METHOD PROTECTED OnExecute
VAR
END_VAR
out.Value := in1.Value AND in2.Value;
END_METHOD

END_FUNCTION_BLOCK

// Logic/Nodes/AND/AND_DINT
{attribute 'linkalways'} 
{attribute 'no_explicit_call' := 'This FB is a CLASS and must be accessed using methods or properties'}
{attribute 'enable_dynamic_creation'}
FUNCTION_BLOCK FINAL AND_DINT EXTENDS Node
VAR
	in1 : _DINT(0);
	in2 : _DINT(0);
	out : _DINT(0);
END_VAR

METHOD FB_init : BOOL
VAR_INPUT
	bInitRetains : BOOL; // if TRUE, the retain variables are initialized (warm start / cold start)
	bInCopyCode : BOOL;  // if TRUE, the instance afterwards gets moved into the copy code (online change)
END_VAR
AddInput('in1',THIS^.in1);
AddInput('in2',THIS^.in2);
AddOutput('out', THIS^.out);
END_METHOD

METHOD PUBLIC Clone : I_Node
VAR
	pNode : POINTER TO AND_DINT;
END_VAR
pNode := __NEW(AND_DINT);
Clone := pNode^;
END_METHOD

METHOD PROTECTED OnExecute
VAR
END_VAR
out.Value := in1.Value AND in2.Value;
END_METHOD

END_FUNCTION_BLOCK

// Logic/Nodes/AND/AND_DWORD
{attribute 'linkalways'} 
{attribute 'no_explicit_call' := 'This FB is a CLASS and must be accessed using methods or properties'}
{attribute 'enable_dynamic_creation'}
FUNCTION_BLOCK FINAL AND_DWORD EXTENDS Node
VAR
	in1 : _DWORD(0);
	in2 : _DWORD(0);
	out : _DWORD(0);
END_VAR

METHOD FB_init : BOOL
VAR_INPUT
	bInitRetains : BOOL; // if TRUE, the retain variables are initialized (warm start / cold start)
	bInCopyCode : BOOL;  // if TRUE, the instance afterwards gets moved into the copy code (online change)
END_VAR
AddInput('in1',THIS^.in1);
AddInput('in2',THIS^.in2);
AddOutput('out', THIS^.out);
END_METHOD

METHOD PUBLIC Clone : I_Node
VAR
	pNode : POINTER TO AND_DWORD;
END_VAR
pNode := __NEW(AND_DWORD);
Clone := pNode^;
END_METHOD

METHOD PROTECTED OnExecute
VAR
END_VAR
out.Value := in1.Value AND in2.Value;
END_METHOD

END_FUNCTION_BLOCK

// Logic/Nodes/AND/AND_INT
{attribute 'linkalways'} 
{attribute 'no_explicit_call' := 'This FB is a CLASS and must be accessed using methods or properties'}
{attribute 'enable_dynamic_creation'}
FUNCTION_BLOCK FINAL AND_INT EXTENDS Node
VAR
	in1 : _INT(0);
	in2 : _INT(0);
	out : _INT(0);
END_VAR

METHOD FB_init : BOOL
VAR_INPUT
	bInitRetains : BOOL; // if TRUE, the retain variables are initialized (warm start / cold start)
	bInCopyCode : BOOL;  // if TRUE, the instance afterwards gets moved into the copy code (online change)
END_VAR
AddInput('in1',THIS^.in1);
AddInput('in2',THIS^.in2);
AddOutput('out', THIS^.out);
END_METHOD

METHOD PUBLIC Clone : I_Node
VAR
	pNode : POINTER TO AND_INT;
END_VAR
pNode := __NEW(AND_INT);
Clone := pNode^;
END_METHOD

METHOD PROTECTED OnExecute
VAR
END_VAR
out.Value := in1.Value AND in2.Value;
END_METHOD

END_FUNCTION_BLOCK

// Logic/Nodes/AND/AND_LINT
{attribute 'linkalways'} 
{attribute 'no_explicit_call' := 'This FB is a CLASS and must be accessed using methods or properties'}
{attribute 'enable_dynamic_creation'}
FUNCTION_BLOCK FINAL AND_LINT EXTENDS Node
VAR
	in1 : _LINT(0);
	in2 : _LINT(0);
	out : _LINT(0);
END_VAR

METHOD FB_init : BOOL
VAR_INPUT
	bInitRetains : BOOL; // if TRUE, the retain variables are initialized (warm start / cold start)
	bInCopyCode : BOOL;  // if TRUE, the instance afterwards gets moved into the copy code (online change)
END_VAR
AddInput('in1',THIS^.in1);
AddInput('in2',THIS^.in2);
AddOutput('out', THIS^.out);
END_METHOD

METHOD PUBLIC Clone : I_Node
VAR
	pNode : POINTER TO AND_LINT;
END_VAR
pNode := __NEW(AND_LINT);
Clone := pNode^;
END_METHOD

METHOD PROTECTED OnExecute
VAR
END_VAR
out.Value := in1.Value AND in2.Value;
END_METHOD

END_FUNCTION_BLOCK

// Logic/Nodes/AND/AND_LWORD
{attribute 'linkalways'} 
{attribute 'no_explicit_call' := 'This FB is a CLASS and must be accessed using methods or properties'}
{attribute 'enable_dynamic_creation'}
FUNCTION_BLOCK FINAL AND_LWORD EXTENDS Node
VAR
	in1 : _LWORD(0);
	in2 : _LWORD(0);
	out : _LWORD(0);
END_VAR

METHOD FB_init : BOOL
VAR_INPUT
	bInitRetains : BOOL; // if TRUE, the retain variables are initialized (warm start / cold start)
	bInCopyCode : BOOL;  // if TRUE, the instance afterwards gets moved into the copy code (online change)
END_VAR
AddInput('in1',THIS^.in1);
AddInput('in2',THIS^.in2);
AddOutput('out', THIS^.out);
END_METHOD

METHOD PUBLIC Clone : I_Node
VAR
	pNode : POINTER TO AND_LWORD;
END_VAR
pNode := __NEW(AND_LWORD);
Clone := pNode^;
END_METHOD

METHOD PROTECTED OnExecute
VAR
END_VAR
out.Value := in1.Value AND in2.Value;
END_METHOD

END_FUNCTION_BLOCK

// Logic/Nodes/AND/AND_SINT
{attribute 'linkalways'} 
{attribute 'no_explicit_call' := 'This FB is a CLASS and must be accessed using methods or properties'}
{attribute 'enable_dynamic_creation'}
FUNCTION_BLOCK FINAL AND_SINT EXTENDS Node
VAR
	in1 : _SINT(0);
	in2 : _SINT(0);
	out : _SINT(0);
END_VAR

METHOD FB_init : BOOL
VAR_INPUT
	bInitRetains : BOOL; // if TRUE, the retain variables are initialized (warm start / cold start)
	bInCopyCode : BOOL;  // if TRUE, the instance afterwards gets moved into the copy code (online change)
END_VAR
AddInput('in1',THIS^.in1);
AddInput('in2',THIS^.in2);
AddOutput('out', THIS^.out);
END_METHOD

METHOD PUBLIC Clone : I_Node
VAR
	pNode : POINTER TO AND_SINT;
END_VAR
pNode := __NEW(AND_SINT);
Clone := pNode^;
END_METHOD

METHOD PROTECTED OnExecute
VAR
END_VAR
out.Value := in1.Value AND in2.Value;
END_METHOD

END_FUNCTION_BLOCK

// Logic/Nodes/AND/AND_UDINT
{attribute 'linkalways'} 
{attribute 'no_explicit_call' := 'This FB is a CLASS and must be accessed using methods or properties'}
{attribute 'enable_dynamic_creation'}
FUNCTION_BLOCK FINAL AND_UDINT EXTENDS Node
VAR
	in1 : _UDINT(0);
	in2 : _UDINT(0);
	out : _UDINT(0);
END_VAR

METHOD FB_init : BOOL
VAR_INPUT
	bInitRetains : BOOL; // if TRUE, the retain variables are initialized (warm start / cold start)
	bInCopyCode : BOOL;  // if TRUE, the instance afterwards gets moved into the copy code (online change)
END_VAR
AddInput('in1',THIS^.in1);
AddInput('in2',THIS^.in2);
AddOutput('out', THIS^.out);
END_METHOD

METHOD PUBLIC Clone : I_Node
VAR
	pNode : POINTER TO AND_UDINT;
END_VAR
pNode := __NEW(AND_UDINT);
Clone := pNode^;
END_METHOD

METHOD PROTECTED OnExecute
VAR
END_VAR
out.Value := in1.Value AND in2.Value;
END_METHOD

END_FUNCTION_BLOCK

// Logic/Nodes/AND/AND_UINT
{attribute 'linkalways'} 
{attribute 'no_explicit_call' := 'This FB is a CLASS and must be accessed using methods or properties'}
{attribute 'enable_dynamic_creation'}
FUNCTION_BLOCK FINAL AND_UINT EXTENDS Node
VAR
	in1 : _UINT(0);
	in2 : _UINT(0);
	out : _UINT(0);
END_VAR

METHOD FB_init : BOOL
VAR_INPUT
	bInitRetains : BOOL; // if TRUE, the retain variables are initialized (warm start / cold start)
	bInCopyCode : BOOL;  // if TRUE, the instance afterwards gets moved into the copy code (online change)
END_VAR
AddInput('in1',THIS^.in1);
AddInput('in2',THIS^.in2);
AddOutput('out', THIS^.out);
END_METHOD

METHOD PUBLIC Clone : I_Node
VAR
	pNode : POINTER TO AND_UINT;
END_VAR
pNode := __NEW(AND_UINT);
Clone := pNode^;
END_METHOD

METHOD PROTECTED OnExecute
VAR
END_VAR
out.Value := in1.Value AND in2.Value;
END_METHOD

END_FUNCTION_BLOCK

// Logic/Nodes/AND/AND_ULINT
{attribute 'linkalways'} 
{attribute 'no_explicit_call' := 'This FB is a CLASS and must be accessed using methods or properties'}
{attribute 'enable_dynamic_creation'}
FUNCTION_BLOCK FINAL AND_ULINT EXTENDS Node
VAR
	in1 : _ULINT(0);
	in2 : _ULINT(0);
	out : _ULINT(0);
END_VAR

METHOD FB_init : BOOL
VAR_INPUT
	bInitRetains : BOOL; // if TRUE, the retain variables are initialized (warm start / cold start)
	bInCopyCode : BOOL;  // if TRUE, the instance afterwards gets moved into the copy code (online change)
END_VAR
AddInput('in1',THIS^.in1);
AddInput('in2',THIS^.in2);
AddOutput('out', THIS^.out);
END_METHOD

METHOD PUBLIC Clone : I_Node
VAR
	pNode : POINTER TO AND_ULINT;
END_VAR
pNode := __NEW(AND_ULINT);
Clone := pNode^;
END_METHOD

METHOD PROTECTED OnExecute
VAR
END_VAR
out.Value := in1.Value AND in2.Value;
END_METHOD

END_FUNCTION_BLOCK

// Logic/Nodes/AND/AND_USINT
{attribute 'linkalways'} 
{attribute 'no_explicit_call' := 'This FB is a CLASS and must be accessed using methods or properties'}
{attribute 'enable_dynamic_creation'}
FUNCTION_BLOCK FINAL AND_USINT EXTENDS Node
VAR
	in1 : _USINT(0);
	in2 : _USINT(0);
	out : _USINT(0);
END_VAR

METHOD FB_init : BOOL
VAR_INPUT
	bInitRetains : BOOL; // if TRUE, the retain variables are initialized (warm start / cold start)
	bInCopyCode : BOOL;  // if TRUE, the instance afterwards gets moved into the copy code (online change)
END_VAR
AddInput('in1',THIS^.in1);
AddInput('in2',THIS^.in2);
AddOutput('out', THIS^.out);
END_METHOD

METHOD PUBLIC Clone : I_Node
VAR
	pNode : POINTER TO AND_USINT;
END_VAR
pNode := __NEW(AND_USINT);
Clone := pNode^;
END_METHOD

METHOD PROTECTED OnExecute
VAR
END_VAR
out.Value := in1.Value AND in2.Value;
END_METHOD

END_FUNCTION_BLOCK

// Logic/Nodes/AND/AND_WORD
{attribute 'linkalways'} 
{attribute 'no_explicit_call' := 'This FB is a CLASS and must be accessed using methods or properties'}
{attribute 'enable_dynamic_creation'}
FUNCTION_BLOCK FINAL AND_WORD EXTENDS Node
VAR
	in1 : _WORD(0);
	in2 : _WORD(0);
	out : _WORD(0);
END_VAR

METHOD FB_init : BOOL
VAR_INPUT
	bInitRetains : BOOL; // if TRUE, the retain variables are initialized (warm start / cold start)
	bInCopyCode : BOOL;  // if TRUE, the instance afterwards gets moved into the copy code (online change)
END_VAR
AddInput('in1',THIS^.in1);
AddInput('in2',THIS^.in2);
AddOutput('out', THIS^.out);
END_METHOD

METHOD PUBLIC Clone : I_Node
VAR
	pNode : POINTER TO AND_WORD;
END_VAR
pNode := __NEW(AND_WORD);
Clone := pNode^;
END_METHOD

METHOD PROTECTED OnExecute
VAR
END_VAR
out.Value := in1.Value AND in2.Value;
END_METHOD

END_FUNCTION_BLOCK

// Logic/Nodes/NOT/NOT_BOOL
{attribute 'linkalways'} 
{attribute 'no_explicit_call' := 'This FB is a CLASS and must be accessed using methods or properties'}
{attribute 'enable_dynamic_creation'}
FUNCTION_BLOCK FINAL NOT_BOOL EXTENDS Node
VAR
	in : _BOOL(FALSE);
	out : _BOOL(FALSE);
END_VAR

METHOD FB_init : BOOL
VAR_INPUT
	bInitRetains : BOOL; // if TRUE, the retain variables are initialized (warm start / cold start)
	bInCopyCode : BOOL;  // if TRUE, the instance afterwards gets moved into the copy code (online change)
END_VAR
AddInput('in',THIS^.in);
AddOutput('out', THIS^.out);
END_METHOD

METHOD PUBLIC Clone : I_Node
VAR
	pNode : POINTER TO NOT_BOOL;
END_VAR
pNode := __NEW(NOT_BOOL);
Clone := pNode^;
END_METHOD

METHOD PROTECTED OnExecute
VAR
END_VAR
out.Value := NOT in.Value;
END_METHOD

END_FUNCTION_BLOCK

// Logic/Nodes/NOT/NOT_BYTE
{attribute 'linkalways'} 
{attribute 'no_explicit_call' := 'This FB is a CLASS and must be accessed using methods or properties'}
{attribute 'enable_dynamic_creation'}
FUNCTION_BLOCK FINAL NOT_BYTE EXTENDS Node
VAR
	in : _BYTE(0);
	out : _BYTE(0);
END_VAR

METHOD FB_init : BOOL
VAR_INPUT
	bInitRetains : BOOL; // if TRUE, the retain variables are initialized (warm start / cold start)
	bInCopyCode : BOOL;  // if TRUE, the instance afterwards gets moved into the copy code (online change)
END_VAR
AddInput('in',THIS^.in);
AddOutput('out', THIS^.out);
END_METHOD

METHOD PUBLIC Clone : I_Node
VAR
	pNode : POINTER TO NOT_BYTE;
END_VAR
pNode := __NEW(NOT_BYTE);
Clone := pNode^;
END_METHOD

METHOD PROTECTED OnExecute
VAR
END_VAR
out.Value := NOT in.Value;
END_METHOD

END_FUNCTION_BLOCK

// Logic/Nodes/NOT/NOT_DINT
{attribute 'linkalways'} 
{attribute 'no_explicit_call' := 'This FB is a CLASS and must be accessed using methods or properties'}
{attribute 'enable_dynamic_creation'}
FUNCTION_BLOCK FINAL NOT_DINT EXTENDS Node
VAR
	in : _DINT(0);
	out : _DINT(0);
END_VAR

METHOD FB_init : BOOL
VAR_INPUT
	bInitRetains : BOOL; // if TRUE, the retain variables are initialized (warm start / cold start)
	bInCopyCode : BOOL;  // if TRUE, the instance afterwards gets moved into the copy code (online change)
END_VAR
AddInput('in',THIS^.in);
AddOutput('out', THIS^.out);
END_METHOD

METHOD PUBLIC Clone : I_Node
VAR
	pNode : POINTER TO NOT_DINT;
END_VAR
pNode := __NEW(NOT_DINT);
Clone := pNode^;
END_METHOD

METHOD PROTECTED OnExecute
VAR
END_VAR
out.Value := NOT in.Value;
END_METHOD

END_FUNCTION_BLOCK

// Logic/Nodes/NOT/NOT_DWORD
{attribute 'linkalways'} 
{attribute 'no_explicit_call' := 'This FB is a CLASS and must be accessed using methods or properties'}
{attribute 'enable_dynamic_creation'}
FUNCTION_BLOCK FINAL NOT_DWORD EXTENDS Node
VAR
	in : _DWORD(0);
	out : _DWORD(0);
END_VAR

METHOD FB_init : BOOL
VAR_INPUT
	bInitRetains : BOOL; // if TRUE, the retain variables are initialized (warm start / cold start)
	bInCopyCode : BOOL;  // if TRUE, the instance afterwards gets moved into the copy code (online change)
END_VAR
AddInput('in',THIS^.in);
AddOutput('out', THIS^.out);
END_METHOD

METHOD PUBLIC Clone : I_Node
VAR
	pNode : POINTER TO NOT_DWORD;
END_VAR
pNode := __NEW(NOT_DWORD);
Clone := pNode^;
END_METHOD

METHOD PROTECTED OnExecute
VAR
END_VAR
out.Value := NOT in.Value;
END_METHOD

END_FUNCTION_BLOCK

// Logic/Nodes/NOT/NOT_INT
{attribute 'linkalways'} 
{attribute 'no_explicit_call' := 'This FB is a CLASS and must be accessed using methods or properties'}
{attribute 'enable_dynamic_creation'}
FUNCTION_BLOCK FINAL NOT_INT EXTENDS Node
VAR
	in : _INT(0);
	out : _INT(0);
END_VAR

METHOD FB_init : BOOL
VAR_INPUT
	bInitRetains : BOOL; // if TRUE, the retain variables are initialized (warm start / cold start)
	bInCopyCode : BOOL;  // if TRUE, the instance afterwards gets moved into the copy code (online change)
END_VAR
AddInput('in',THIS^.in);
AddOutput('out', THIS^.out);
END_METHOD

METHOD PUBLIC Clone : I_Node
VAR
	pNode : POINTER TO NOT_INT;
END_VAR
pNode := __NEW(NOT_INT);
Clone := pNode^;
END_METHOD

METHOD PROTECTED OnExecute
VAR
END_VAR
out.Value := NOT in.Value;
END_METHOD

END_FUNCTION_BLOCK

// Logic/Nodes/NOT/NOT_LINT
{attribute 'linkalways'} 
{attribute 'no_explicit_call' := 'This FB is a CLASS and must be accessed using methods or properties'}
{attribute 'enable_dynamic_creation'}
FUNCTION_BLOCK FINAL NOT_LINT EXTENDS Node
VAR
	in : _LINT(0);
	out : _LINT(0);
END_VAR

METHOD FB_init : BOOL
VAR_INPUT
	bInitRetains : BOOL; // if TRUE, the retain variables are initialized (warm start / cold start)
	bInCopyCode : BOOL;  // if TRUE, the instance afterwards gets moved into the copy code (online change)
END_VAR
AddInput('in',THIS^.in);
AddOutput('out', THIS^.out);
END_METHOD

METHOD PUBLIC Clone : I_Node
VAR
	pNode : POINTER TO NOT_LINT;
END_VAR
pNode := __NEW(NOT_LINT);
Clone := pNode^;
END_METHOD

METHOD PROTECTED OnExecute
VAR
END_VAR
out.Value := NOT in.Value;
END_METHOD

END_FUNCTION_BLOCK

// Logic/Nodes/NOT/NOT_LWORD
{attribute 'linkalways'} 
{attribute 'no_explicit_call' := 'This FB is a CLASS and must be accessed using methods or properties'}
{attribute 'enable_dynamic_creation'}
FUNCTION_BLOCK FINAL NOT_LWORD EXTENDS Node
VAR
	in : _LWORD(0);
	out : _LWORD(0);
END_VAR

METHOD FB_init : BOOL
VAR_INPUT
	bInitRetains : BOOL; // if TRUE, the retain variables are initialized (warm start / cold start)
	bInCopyCode : BOOL;  // if TRUE, the instance afterwards gets moved into the copy code (online change)
END_VAR
AddInput('in',THIS^.in);
AddOutput('out', THIS^.out);
END_METHOD

METHOD PUBLIC Clone : I_Node
VAR
	pNode : POINTER TO NOT_LWORD;
END_VAR
pNode := __NEW(NOT_LWORD);
Clone := pNode^;
END_METHOD

METHOD PROTECTED OnExecute
VAR
END_VAR
out.Value := NOT in.Value;
END_METHOD

END_FUNCTION_BLOCK

// Logic/Nodes/NOT/NOT_SINT
{attribute 'linkalways'} 
{attribute 'no_explicit_call' := 'This FB is a CLASS and must be accessed using methods or properties'}
{attribute 'enable_dynamic_creation'}
FUNCTION_BLOCK FINAL NOT_SINT EXTENDS Node
VAR
	in : _SINT(0);
	out : _SINT(0);
END_VAR

METHOD FB_init : BOOL
VAR_INPUT
	bInitRetains : BOOL; // if TRUE, the retain variables are initialized (warm start / cold start)
	bInCopyCode : BOOL;  // if TRUE, the instance afterwards gets moved into the copy code (online change)
END_VAR
AddInput('in',THIS^.in);
AddOutput('out', THIS^.out);
END_METHOD

METHOD PUBLIC Clone : I_Node
VAR
	pNode : POINTER TO NOT_SINT;
END_VAR
pNode := __NEW(NOT_SINT);
Clone := pNode^;
END_METHOD

METHOD PROTECTED OnExecute
VAR
END_VAR
out.Value := NOT in.Value;
END_METHOD

END_FUNCTION_BLOCK

// Logic/Nodes/NOT/NOT_UDINT
{attribute 'linkalways'} 
{attribute 'no_explicit_call' := 'This FB is a CLASS and must be accessed using methods or properties'}
{attribute 'enable_dynamic_creation'}
FUNCTION_BLOCK FINAL NOT_UDINT EXTENDS Node
VAR
	in : _UDINT(0);
	out : _UDINT(0);
END_VAR

METHOD FB_init : BOOL
VAR_INPUT
	bInitRetains : BOOL; // if TRUE, the retain variables are initialized (warm start / cold start)
	bInCopyCode : BOOL;  // if TRUE, the instance afterwards gets moved into the copy code (online change)
END_VAR
AddInput('in',THIS^.in);
AddOutput('out', THIS^.out);
END_METHOD

METHOD PUBLIC Clone : I_Node
VAR
	pNode : POINTER TO NOT_UDINT;
END_VAR
pNode := __NEW(NOT_UDINT);
Clone := pNode^;
END_METHOD

METHOD PROTECTED OnExecute
VAR
END_VAR
out.Value := NOT in.Value;
END_METHOD

END_FUNCTION_BLOCK

// Logic/Nodes/NOT/NOT_UINT
{attribute 'linkalways'} 
{attribute 'no_explicit_call' := 'This FB is a CLASS and must be accessed using methods or properties'}
{attribute 'enable_dynamic_creation'}
FUNCTION_BLOCK FINAL NOT_UINT EXTENDS Node
VAR
	in : _UINT(0);
	out : _UINT(0);
END_VAR

METHOD FB_init : BOOL
VAR_INPUT
	bInitRetains : BOOL; // if TRUE, the retain variables are initialized (warm start / cold start)
	bInCopyCode : BOOL;  // if TRUE, the instance afterwards gets moved into the copy code (online change)
END_VAR
AddInput('in',THIS^.in);
AddOutput('out', THIS^.out);
END_METHOD

METHOD PUBLIC Clone : I_Node
VAR
	pNode : POINTER TO NOT_UINT;
END_VAR
pNode := __NEW(NOT_UINT);
Clone := pNode^;
END_METHOD

METHOD PROTECTED OnExecute
VAR
END_VAR
out.Value := NOT in.Value;
END_METHOD

END_FUNCTION_BLOCK

// Logic/Nodes/NOT/NOT_ULINT
{attribute 'linkalways'} 
{attribute 'no_explicit_call' := 'This FB is a CLASS and must be accessed using methods or properties'}
{attribute 'enable_dynamic_creation'}
FUNCTION_BLOCK FINAL NOT_ULINT EXTENDS Node
VAR
	in : _ULINT(0);
	out : _ULINT(0);
END_VAR

METHOD FB_init : BOOL
VAR_INPUT
	bInitRetains : BOOL; // if TRUE, the retain variables are initialized (warm start / cold start)
	bInCopyCode : BOOL;  // if TRUE, the instance afterwards gets moved into the copy code (online change)
END_VAR
AddInput('in',THIS^.in);
AddOutput('out', THIS^.out);
END_METHOD

METHOD PUBLIC Clone : I_Node
VAR
	pNode : POINTER TO NOT_ULINT;
END_VAR
pNode := __NEW(NOT_ULINT);
Clone := pNode^;
END_METHOD

METHOD PROTECTED OnExecute
VAR
END_VAR
out.Value := NOT in.Value;
END_METHOD

END_FUNCTION_BLOCK

// Logic/Nodes/NOT/NOT_USINT
{attribute 'linkalways'} 
{attribute 'no_explicit_call' := 'This FB is a CLASS and must be accessed using methods or properties'}
{attribute 'enable_dynamic_creation'}
FUNCTION_BLOCK FINAL NOT_USINT EXTENDS Node
VAR
	in : _USINT(0);
	out : _USINT(0);
END_VAR

METHOD FB_init : BOOL
VAR_INPUT
	bInitRetains : BOOL; // if TRUE, the retain variables are initialized (warm start / cold start)
	bInCopyCode : BOOL;  // if TRUE, the instance afterwards gets moved into the copy code (online change)
END_VAR
AddInput('in',THIS^.in);
AddOutput('out', THIS^.out);
END_METHOD

METHOD PUBLIC Clone : I_Node
VAR
	pNode : POINTER TO NOT_USINT;
END_VAR
pNode := __NEW(NOT_USINT);
Clone := pNode^;
END_METHOD

METHOD PROTECTED OnExecute
VAR
END_VAR
out.Value := NOT in.Value;
END_METHOD

END_FUNCTION_BLOCK

// Logic/Nodes/NOT/NOT_WORD
{attribute 'linkalways'} 
{attribute 'no_explicit_call' := 'This FB is a CLASS and must be accessed using methods or properties'}
{attribute 'enable_dynamic_creation'}
FUNCTION_BLOCK FINAL NOT_WORD EXTENDS Node
VAR
	in : _WORD(0);
	out : _WORD(0);
END_VAR

METHOD FB_init : BOOL
VAR_INPUT
	bInitRetains : BOOL; // if TRUE, the retain variables are initialized (warm start / cold start)
	bInCopyCode : BOOL;  // if TRUE, the instance afterwards gets moved into the copy code (online change)
END_VAR
AddInput('in',THIS^.in);
AddOutput('out', THIS^.out);
END_METHOD

METHOD PUBLIC Clone : I_Node
VAR
	pNode : POINTER TO NOT_WORD;
END_VAR
pNode := __NEW(NOT_WORD);
Clone := pNode^;
END_METHOD

METHOD PROTECTED OnExecute
VAR
END_VAR
out.Value := NOT in.Value;
END_METHOD

END_FUNCTION_BLOCK

// Logic/Nodes/OR/OR_BOOL
{attribute 'linkalways'} 
{attribute 'no_explicit_call' := 'This FB is a CLASS and must be accessed using methods or properties'}
{attribute 'enable_dynamic_creation'}
FUNCTION_BLOCK FINAL OR_BOOL EXTENDS Node
VAR
	in1 : _BOOL(FALSE);
	in2 : _BOOL(FALSE);
	out : _BOOL(FALSE);
END_VAR

METHOD FB_init : BOOL
VAR_INPUT
	bInitRetains : BOOL; // if TRUE, the retain variables are initialized (warm start / cold start)
	bInCopyCode : BOOL;  // if TRUE, the instance afterwards gets moved into the copy code (online change)
END_VAR
AddInput('in1',THIS^.in1);
AddInput('in2',THIS^.in2);
AddOutput('out', THIS^.out);
END_METHOD

METHOD PUBLIC Clone : I_Node
VAR
	pNode : POINTER TO OR_BOOL;
END_VAR
pNode := __NEW(OR_BOOL);
Clone := pNode^;
END_METHOD

METHOD PROTECTED OnExecute
VAR
END_VAR
out.Value := in1.Value OR in2.Value;
END_METHOD

END_FUNCTION_BLOCK

// Logic/Nodes/OR/OR_BYTE
{attribute 'linkalways'} 
{attribute 'no_explicit_call' := 'This FB is a CLASS and must be accessed using methods or properties'}
{attribute 'enable_dynamic_creation'}
FUNCTION_BLOCK FINAL OR_BYTE EXTENDS Node
VAR
	in1 : _BYTE(0);
	in2 : _BYTE(0);
	out : _BYTE(0);
END_VAR

METHOD FB_init : BOOL
VAR_INPUT
	bInitRetains : BOOL; // if TRUE, the retain variables are initialized (warm start / cold start)
	bInCopyCode : BOOL;  // if TRUE, the instance afterwards gets moved into the copy code (online change)
END_VAR
AddInput('in1',THIS^.in1);
AddInput('in2',THIS^.in2);
AddOutput('out', THIS^.out);
END_METHOD

METHOD PUBLIC Clone : I_Node
VAR
	pNode : POINTER TO OR_BYTE;
END_VAR
pNode := __NEW(OR_BYTE);
Clone := pNode^;
END_METHOD

METHOD PROTECTED OnExecute
VAR
END_VAR
out.Value := in1.Value OR in2.Value;
END_METHOD

END_FUNCTION_BLOCK

// Logic/Nodes/OR/OR_DINT
{attribute 'linkalways'} 
{attribute 'no_explicit_call' := 'This FB is a CLASS and must be accessed using methods or properties'}
{attribute 'enable_dynamic_creation'}
FUNCTION_BLOCK FINAL OR_DINT EXTENDS Node
VAR
	in1 : _DINT(0);
	in2 : _DINT(0);
	out : _DINT(0);
END_VAR

METHOD FB_init : BOOL
VAR_INPUT
	bInitRetains : BOOL; // if TRUE, the retain variables are initialized (warm start / cold start)
	bInCopyCode : BOOL;  // if TRUE, the instance afterwards gets moved into the copy code (online change)
END_VAR
AddInput('in1',THIS^.in1);
AddInput('in2',THIS^.in2);
AddOutput('out', THIS^.out);
END_METHOD

METHOD PUBLIC Clone : I_Node
VAR
	pNode : POINTER TO OR_DINT;
END_VAR
pNode := __NEW(OR_DINT);
Clone := pNode^;
END_METHOD

METHOD PROTECTED OnExecute
VAR
END_VAR
out.Value := in1.Value OR in2.Value;
END_METHOD

END_FUNCTION_BLOCK

// Logic/Nodes/OR/OR_DWORD
{attribute 'linkalways'} 
{attribute 'no_explicit_call' := 'This FB is a CLASS and must be accessed using methods or properties'}
{attribute 'enable_dynamic_creation'}
FUNCTION_BLOCK FINAL OR_DWORD EXTENDS Node
VAR
	in1 : _DWORD(0);
	in2 : _DWORD(0);
	out : _DWORD(0);
END_VAR

METHOD FB_init : BOOL
VAR_INPUT
	bInitRetains : BOOL; // if TRUE, the retain variables are initialized (warm start / cold start)
	bInCopyCode : BOOL;  // if TRUE, the instance afterwards gets moved into the copy code (online change)
END_VAR
AddInput('in1',THIS^.in1);
AddInput('in2',THIS^.in2);
AddOutput('out', THIS^.out);
END_METHOD

METHOD PUBLIC Clone : I_Node
VAR
	pNode : POINTER TO OR_DWORD;
END_VAR
pNode := __NEW(OR_DWORD);
Clone := pNode^;
END_METHOD

METHOD PROTECTED OnExecute
VAR
END_VAR
out.Value := in1.Value OR in2.Value;
END_METHOD

END_FUNCTION_BLOCK

// Logic/Nodes/OR/OR_INT
{attribute 'linkalways'} 
{attribute 'no_explicit_call' := 'This FB is a CLASS and must be accessed using methods or properties'}
{attribute 'enable_dynamic_creation'}
FUNCTION_BLOCK FINAL OR_INT EXTENDS Node
VAR
	in1 : _INT(0);
	in2 : _INT(0);
	out : _INT(0);
END_VAR

METHOD FB_init : BOOL
VAR_INPUT
	bInitRetains : BOOL; // if TRUE, the retain variables are initialized (warm start / cold start)
	bInCopyCode : BOOL;  // if TRUE, the instance afterwards gets moved into the copy code (online change)
END_VAR
AddInput('in1',THIS^.in1);
AddInput('in2',THIS^.in2);
AddOutput('out', THIS^.out);
END_METHOD

METHOD PUBLIC Clone : I_Node
VAR
	pNode : POINTER TO OR_INT;
END_VAR
pNode := __NEW(OR_INT);
Clone := pNode^;
END_METHOD

METHOD PROTECTED OnExecute
VAR
END_VAR
out.Value := in1.Value OR in2.Value;
END_METHOD

END_FUNCTION_BLOCK

// Logic/Nodes/OR/OR_LINT
{attribute 'linkalways'} 
{attribute 'no_explicit_call' := 'This FB is a CLASS and must be accessed using methods or properties'}
{attribute 'enable_dynamic_creation'}
FUNCTION_BLOCK FINAL OR_LINT EXTENDS Node
VAR
	in1 : _LINT(0);
	in2 : _LINT(0);
	out : _LINT(0);
END_VAR

METHOD FB_init : BOOL
VAR_INPUT
	bInitRetains : BOOL; // if TRUE, the retain variables are initialized (warm start / cold start)
	bInCopyCode : BOOL;  // if TRUE, the instance afterwards gets moved into the copy code (online change)
END_VAR
AddInput('in1',THIS^.in1);
AddInput('in2',THIS^.in2);
AddOutput('out', THIS^.out);
END_METHOD

METHOD PUBLIC Clone : I_Node
VAR
	pNode : POINTER TO OR_LINT;
END_VAR
pNode := __NEW(OR_LINT);
Clone := pNode^;
END_METHOD

METHOD PROTECTED OnExecute
VAR
END_VAR
out.Value := in1.Value OR in2.Value;
END_METHOD

END_FUNCTION_BLOCK

// Logic/Nodes/OR/OR_LWORD
{attribute 'linkalways'} 
{attribute 'no_explicit_call' := 'This FB is a CLASS and must be accessed using methods or properties'}
{attribute 'enable_dynamic_creation'}
FUNCTION_BLOCK FINAL OR_LWORD EXTENDS Node
VAR
	in1 : _LWORD(0);
	in2 : _LWORD(0);
	out : _LWORD(0);
END_VAR

METHOD FB_init : BOOL
VAR_INPUT
	bInitRetains : BOOL; // if TRUE, the retain variables are initialized (warm start / cold start)
	bInCopyCode : BOOL;  // if TRUE, the instance afterwards gets moved into the copy code (online change)
END_VAR
AddInput('in1',THIS^.in1);
AddInput('in2',THIS^.in2);
AddOutput('out', THIS^.out);
END_METHOD

METHOD PUBLIC Clone : I_Node
VAR
	pNode : POINTER TO OR_LWORD;
END_VAR
pNode := __NEW(OR_LWORD);
Clone := pNode^;
END_METHOD

METHOD PROTECTED OnExecute
VAR
END_VAR
out.Value := in1.Value OR in2.Value;
END_METHOD

END_FUNCTION_BLOCK

// Logic/Nodes/OR/OR_SINT
{attribute 'linkalways'} 
{attribute 'no_explicit_call' := 'This FB is a CLASS and must be accessed using methods or properties'}
{attribute 'enable_dynamic_creation'}
FUNCTION_BLOCK FINAL OR_SINT EXTENDS Node
VAR
	in1 : _SINT(0);
	in2 : _SINT(0);
	out : _SINT(0);
END_VAR

METHOD FB_init : BOOL
VAR_INPUT
	bInitRetains : BOOL; // if TRUE, the retain variables are initialized (warm start / cold start)
	bInCopyCode : BOOL;  // if TRUE, the instance afterwards gets moved into the copy code (online change)
END_VAR
AddInput('in1',THIS^.in1);
AddInput('in2',THIS^.in2);
AddOutput('out', THIS^.out);
END_METHOD

METHOD PUBLIC Clone : I_Node
VAR
	pNode : POINTER TO OR_SINT;
END_VAR
pNode := __NEW(OR_SINT);
Clone := pNode^;
END_METHOD

METHOD PROTECTED OnExecute
VAR
END_VAR
out.Value := in1.Value OR in2.Value;
END_METHOD

END_FUNCTION_BLOCK

// Logic/Nodes/OR/OR_UDINT
{attribute 'linkalways'} 
{attribute 'no_explicit_call' := 'This FB is a CLASS and must be accessed using methods or properties'}
{attribute 'enable_dynamic_creation'}
FUNCTION_BLOCK FINAL OR_UDINT EXTENDS Node
VAR
	in1 : _UDINT(0);
	in2 : _UDINT(0);
	out : _UDINT(0);
END_VAR

METHOD FB_init : BOOL
VAR_INPUT
	bInitRetains : BOOL; // if TRUE, the retain variables are initialized (warm start / cold start)
	bInCopyCode : BOOL;  // if TRUE, the instance afterwards gets moved into the copy code (online change)
END_VAR
AddInput('in1',THIS^.in1);
AddInput('in2',THIS^.in2);
AddOutput('out', THIS^.out);
END_METHOD

METHOD PUBLIC Clone : I_Node
VAR
	pNode : POINTER TO OR_UDINT;
END_VAR
pNode := __NEW(OR_UDINT);
Clone := pNode^;
END_METHOD

METHOD PROTECTED OnExecute
VAR
END_VAR
out.Value := in1.Value OR in2.Value;
END_METHOD

END_FUNCTION_BLOCK

// Logic/Nodes/OR/OR_UINT
{attribute 'linkalways'} 
{attribute 'no_explicit_call' := 'This FB is a CLASS and must be accessed using methods or properties'}
{attribute 'enable_dynamic_creation'}
FUNCTION_BLOCK FINAL OR_UINT EXTENDS Node
VAR
	in1 : _UINT(0);
	in2 : _UINT(0);
	out : _UINT(0);
END_VAR

METHOD FB_init : BOOL
VAR_INPUT
	bInitRetains : BOOL; // if TRUE, the retain variables are initialized (warm start / cold start)
	bInCopyCode : BOOL;  // if TRUE, the instance afterwards gets moved into the copy code (online change)
END_VAR
AddInput('in1',THIS^.in1);
AddInput('in2',THIS^.in2);
AddOutput('out', THIS^.out);
END_METHOD

METHOD PUBLIC Clone : I_Node
VAR
	pNode : POINTER TO OR_UINT;
END_VAR
pNode := __NEW(OR_UINT);
Clone := pNode^;
END_METHOD

METHOD PROTECTED OnExecute
VAR
END_VAR
out.Value := in1.Value OR in2.Value;
END_METHOD

END_FUNCTION_BLOCK

// Logic/Nodes/OR/OR_ULINT
{attribute 'linkalways'} 
{attribute 'no_explicit_call' := 'This FB is a CLASS and must be accessed using methods or properties'}
{attribute 'enable_dynamic_creation'}
FUNCTION_BLOCK FINAL OR_ULINT EXTENDS Node
VAR
	in1 : _ULINT(0);
	in2 : _ULINT(0);
	out : _ULINT(0);
END_VAR

METHOD FB_init : BOOL
VAR_INPUT
	bInitRetains : BOOL; // if TRUE, the retain variables are initialized (warm start / cold start)
	bInCopyCode : BOOL;  // if TRUE, the instance afterwards gets moved into the copy code (online change)
END_VAR
AddInput('in1',THIS^.in1);
AddInput('in2',THIS^.in2);
AddOutput('out', THIS^.out);
END_METHOD

METHOD PUBLIC Clone : I_Node
VAR
	pNode : POINTER TO OR_ULINT;
END_VAR
pNode := __NEW(OR_ULINT);
Clone := pNode^;
END_METHOD

METHOD PROTECTED OnExecute
VAR
END_VAR
out.Value := in1.Value OR in2.Value;
END_METHOD

END_FUNCTION_BLOCK

// Logic/Nodes/OR/OR_USINT
{attribute 'linkalways'} 
{attribute 'no_explicit_call' := 'This FB is a CLASS and must be accessed using methods or properties'}
{attribute 'enable_dynamic_creation'}
FUNCTION_BLOCK FINAL OR_USINT EXTENDS Node
VAR
	in1 : _USINT(0);
	in2 : _USINT(0);
	out : _USINT(0);
END_VAR

METHOD FB_init : BOOL
VAR_INPUT
	bInitRetains : BOOL; // if TRUE, the retain variables are initialized (warm start / cold start)
	bInCopyCode : BOOL;  // if TRUE, the instance afterwards gets moved into the copy code (online change)
END_VAR
AddInput('in1',THIS^.in1);
AddInput('in2',THIS^.in2);
AddOutput('out', THIS^.out);
END_METHOD

METHOD PUBLIC Clone : I_Node
VAR
	pNode : POINTER TO OR_USINT;
END_VAR
pNode := __NEW(OR_USINT);
Clone := pNode^;
END_METHOD

METHOD PROTECTED OnExecute
VAR
END_VAR
out.Value := in1.Value OR in2.Value;
END_METHOD

END_FUNCTION_BLOCK

// Logic/Nodes/OR/OR_WORD
{attribute 'linkalways'} 
{attribute 'no_explicit_call' := 'This FB is a CLASS and must be accessed using methods or properties'}
{attribute 'enable_dynamic_creation'}
FUNCTION_BLOCK FINAL OR_WORD EXTENDS Node
VAR
	in1 : _WORD(0);
	in2 : _WORD(0);
	out : _WORD(0);
END_VAR

METHOD FB_init : BOOL
VAR_INPUT
	bInitRetains : BOOL; // if TRUE, the retain variables are initialized (warm start / cold start)
	bInCopyCode : BOOL;  // if TRUE, the instance afterwards gets moved into the copy code (online change)
END_VAR
AddInput('in1',THIS^.in1);
AddInput('in2',THIS^.in2);
AddOutput('out', THIS^.out);
END_METHOD

METHOD PUBLIC Clone : I_Node
VAR
	pNode : POINTER TO OR_WORD;
END_VAR
pNode := __NEW(OR_WORD);
Clone := pNode^;
END_METHOD

METHOD PROTECTED OnExecute
VAR
END_VAR
out.Value := in1.Value OR in2.Value;
END_METHOD

END_FUNCTION_BLOCK

// Logic/Nodes/XOR/XOR_BOOL
{attribute 'linkalways'} 
{attribute 'no_explicit_call' := 'This FB is a CLASS and must be accessed using methods or properties'}
{attribute 'enable_dynamic_creation'}
FUNCTION_BLOCK FINAL XOR_BOOL EXTENDS Node
VAR
	in1 : _BOOL(FALSE);
	in2 : _BOOL(FALSE);
	out : _BOOL(FALSE);
END_VAR

METHOD FB_init : BOOL
VAR_INPUT
	bInitRetains : BOOL; // if TRUE, the retain variables are initialized (warm start / cold start)
	bInCopyCode : BOOL;  // if TRUE, the instance afterwards gets moved into the copy code (online change)
END_VAR
AddInput('in1',THIS^.in1);
AddInput('in2',THIS^.in2);
AddOutput('out', THIS^.out);
END_METHOD

METHOD PUBLIC Clone : I_Node
VAR
	pNode : POINTER TO XOR_BOOL;
END_VAR
pNode := __NEW(XOR_BOOL);
Clone := pNode^;
END_METHOD

METHOD PROTECTED OnExecute
VAR
END_VAR
out.Value := in1.Value XOR in2.Value;
END_METHOD

END_FUNCTION_BLOCK

// Logic/Nodes/XOR/XOR_BYTE
{attribute 'linkalways'} 
{attribute 'no_explicit_call' := 'This FB is a CLASS and must be accessed using methods or properties'}
{attribute 'enable_dynamic_creation'}
FUNCTION_BLOCK FINAL XOR_BYTE EXTENDS Node
VAR
	in1 : _BYTE(0);
	in2 : _BYTE(0);
	out : _BYTE(0);
END_VAR

METHOD FB_init : BOOL
VAR_INPUT
	bInitRetains : BOOL; // if TRUE, the retain variables are initialized (warm start / cold start)
	bInCopyCode : BOOL;  // if TRUE, the instance afterwards gets moved into the copy code (online change)
END_VAR
AddInput('in1',THIS^.in1);
AddInput('in2',THIS^.in2);
AddOutput('out', THIS^.out);
END_METHOD

METHOD PUBLIC Clone : I_Node
VAR
	pNode : POINTER TO XOR_BYTE;
END_VAR
pNode := __NEW(XOR_BYTE);
Clone := pNode^;
END_METHOD

METHOD PROTECTED OnExecute
VAR
END_VAR
out.Value := in1.Value XOR in2.Value;
END_METHOD

END_FUNCTION_BLOCK

// Logic/Nodes/XOR/XOR_DINT
{attribute 'linkalways'} 
{attribute 'no_explicit_call' := 'This FB is a CLASS and must be accessed using methods or properties'}
{attribute 'enable_dynamic_creation'}
FUNCTION_BLOCK FINAL XOR_DINT EXTENDS Node
VAR
	in1 : _DINT(0);
	in2 : _DINT(0);
	out : _DINT(0);
END_VAR

METHOD FB_init : BOOL
VAR_INPUT
	bInitRetains : BOOL; // if TRUE, the retain variables are initialized (warm start / cold start)
	bInCopyCode : BOOL;  // if TRUE, the instance afterwards gets moved into the copy code (online change)
END_VAR
AddInput('in1',THIS^.in1);
AddInput('in2',THIS^.in2);
AddOutput('out', THIS^.out);
END_METHOD

METHOD PUBLIC Clone : I_Node
VAR
	pNode : POINTER TO XOR_DINT;
END_VAR
pNode := __NEW(XOR_DINT);
Clone := pNode^;
END_METHOD

METHOD PROTECTED OnExecute
VAR
END_VAR
out.Value := in1.Value XOR in2.Value;
END_METHOD

END_FUNCTION_BLOCK

// Logic/Nodes/XOR/XOR_DWORD
{attribute 'linkalways'} 
{attribute 'no_explicit_call' := 'This FB is a CLASS and must be accessed using methods or properties'}
{attribute 'enable_dynamic_creation'}
FUNCTION_BLOCK FINAL XOR_DWORD EXTENDS Node
VAR
	in1 : _DWORD(0);
	in2 : _DWORD(0);
	out : _DWORD(0);
END_VAR

METHOD FB_init : BOOL
VAR_INPUT
	bInitRetains : BOOL; // if TRUE, the retain variables are initialized (warm start / cold start)
	bInCopyCode : BOOL;  // if TRUE, the instance afterwards gets moved into the copy code (online change)
END_VAR
AddInput('in1',THIS^.in1);
AddInput('in2',THIS^.in2);
AddOutput('out', THIS^.out);
END_METHOD

METHOD PUBLIC Clone : I_Node
VAR
	pNode : POINTER TO XOR_DWORD;
END_VAR
pNode := __NEW(XOR_DWORD);
Clone := pNode^;
END_METHOD

METHOD PROTECTED OnExecute
VAR
END_VAR
out.Value := in1.Value XOR in2.Value;
END_METHOD

END_FUNCTION_BLOCK

// Logic/Nodes/XOR/XOR_INT
{attribute 'linkalways'} 
{attribute 'no_explicit_call' := 'This FB is a CLASS and must be accessed using methods or properties'}
{attribute 'enable_dynamic_creation'}
FUNCTION_BLOCK FINAL XOR_INT EXTENDS Node
VAR
	in1 : _INT(0);
	in2 : _INT(0);
	out : _INT(0);
END_VAR

METHOD FB_init : BOOL
VAR_INPUT
	bInitRetains : BOOL; // if TRUE, the retain variables are initialized (warm start / cold start)
	bInCopyCode : BOOL;  // if TRUE, the instance afterwards gets moved into the copy code (online change)
END_VAR
AddInput('in1',THIS^.in1);
AddInput('in2',THIS^.in2);
AddOutput('out', THIS^.out);
END_METHOD

METHOD PUBLIC Clone : I_Node
VAR
	pNode : POINTER TO XOR_INT;
END_VAR
pNode := __NEW(XOR_INT);
Clone := pNode^;
END_METHOD

METHOD PROTECTED OnExecute
VAR
END_VAR
out.Value := in1.Value XOR in2.Value;
END_METHOD

END_FUNCTION_BLOCK

// Logic/Nodes/XOR/XOR_LINT
{attribute 'linkalways'} 
{attribute 'no_explicit_call' := 'This FB is a CLASS and must be accessed using methods or properties'}
{attribute 'enable_dynamic_creation'}
FUNCTION_BLOCK FINAL XOR_LINT EXTENDS Node
VAR
	in1 : _LINT(0);
	in2 : _LINT(0);
	out : _LINT(0);
END_VAR

METHOD FB_init : BOOL
VAR_INPUT
	bInitRetains : BOOL; // if TRUE, the retain variables are initialized (warm start / cold start)
	bInCopyCode : BOOL;  // if TRUE, the instance afterwards gets moved into the copy code (online change)
END_VAR
AddInput('in1',THIS^.in1);
AddInput('in2',THIS^.in2);
AddOutput('out', THIS^.out);
END_METHOD

METHOD PUBLIC Clone : I_Node
VAR
	pNode : POINTER TO XOR_LINT;
END_VAR
pNode := __NEW(XOR_LINT);
Clone := pNode^;
END_METHOD

METHOD PROTECTED OnExecute
VAR
END_VAR
out.Value := in1.Value XOR in2.Value;
END_METHOD

END_FUNCTION_BLOCK

// Logic/Nodes/XOR/XOR_LWORD
{attribute 'linkalways'} 
{attribute 'no_explicit_call' := 'This FB is a CLASS and must be accessed using methods or properties'}
{attribute 'enable_dynamic_creation'}
FUNCTION_BLOCK FINAL XOR_LWORD EXTENDS Node
VAR
	in1 : _LWORD(0);
	in2 : _LWORD(0);
	out : _LWORD(0);
END_VAR

METHOD FB_init : BOOL
VAR_INPUT
	bInitRetains : BOOL; // if TRUE, the retain variables are initialized (warm start / cold start)
	bInCopyCode : BOOL;  // if TRUE, the instance afterwards gets moved into the copy code (online change)
END_VAR
AddInput('in1',THIS^.in1);
AddInput('in2',THIS^.in2);
AddOutput('out', THIS^.out);
END_METHOD

METHOD PUBLIC Clone : I_Node
VAR
	pNode : POINTER TO XOR_LWORD;
END_VAR
pNode := __NEW(XOR_LWORD);
Clone := pNode^;
END_METHOD

METHOD PROTECTED OnExecute
VAR
END_VAR
out.Value := in1.Value XOR in2.Value;
END_METHOD

END_FUNCTION_BLOCK

// Logic/Nodes/XOR/XOR_SINT
{attribute 'linkalways'} 
{attribute 'no_explicit_call' := 'This FB is a CLASS and must be accessed using methods or properties'}
{attribute 'enable_dynamic_creation'}
FUNCTION_BLOCK FINAL XOR_SINT EXTENDS Node
VAR
	in1 : _SINT(0);
	in2 : _SINT(0);
	out : _SINT(0);
END_VAR

METHOD FB_init : BOOL
VAR_INPUT
	bInitRetains : BOOL; // if TRUE, the retain variables are initialized (warm start / cold start)
	bInCopyCode : BOOL;  // if TRUE, the instance afterwards gets moved into the copy code (online change)
END_VAR
AddInput('in1',THIS^.in1);
AddInput('in2',THIS^.in2);
AddOutput('out', THIS^.out);
END_METHOD

METHOD PUBLIC Clone : I_Node
VAR
	pNode : POINTER TO XOR_SINT;
END_VAR
pNode := __NEW(XOR_SINT);
Clone := pNode^;
END_METHOD

METHOD PROTECTED OnExecute
VAR
END_VAR
out.Value := in1.Value XOR in2.Value;
END_METHOD

END_FUNCTION_BLOCK

// Logic/Nodes/XOR/XOR_UDINT
{attribute 'linkalways'} 
{attribute 'no_explicit_call' := 'This FB is a CLASS and must be accessed using methods or properties'}
{attribute 'enable_dynamic_creation'}
FUNCTION_BLOCK FINAL XOR_UDINT EXTENDS Node
VAR
	in1 : _UDINT(0);
	in2 : _UDINT(0);
	out : _UDINT(0);
END_VAR

METHOD FB_init : BOOL
VAR_INPUT
	bInitRetains : BOOL; // if TRUE, the retain variables are initialized (warm start / cold start)
	bInCopyCode : BOOL;  // if TRUE, the instance afterwards gets moved into the copy code (online change)
END_VAR
AddInput('in1',THIS^.in1);
AddInput('in2',THIS^.in2);
AddOutput('out', THIS^.out);
END_METHOD

METHOD PUBLIC Clone : I_Node
VAR
	pNode : POINTER TO XOR_UDINT;
END_VAR
pNode := __NEW(XOR_UDINT);
Clone := pNode^;
END_METHOD

METHOD PROTECTED OnExecute
VAR
END_VAR
out.Value := in1.Value XOR in2.Value;
END_METHOD

END_FUNCTION_BLOCK

// Logic/Nodes/XOR/XOR_UINT
{attribute 'linkalways'} 
{attribute 'no_explicit_call' := 'This FB is a CLASS and must be accessed using methods or properties'}
{attribute 'enable_dynamic_creation'}
FUNCTION_BLOCK FINAL XOR_UINT EXTENDS Node
VAR
	in1 : _UINT(0);
	in2 : _UINT(0);
	out : _UINT(0);
END_VAR

METHOD FB_init : BOOL
VAR_INPUT
	bInitRetains : BOOL; // if TRUE, the retain variables are initialized (warm start / cold start)
	bInCopyCode : BOOL;  // if TRUE, the instance afterwards gets moved into the copy code (online change)
END_VAR
AddInput('in1',THIS^.in1);
AddInput('in2',THIS^.in2);
AddOutput('out', THIS^.out);
END_METHOD

METHOD PUBLIC Clone : I_Node
VAR
	pNode : POINTER TO XOR_UINT;
END_VAR
pNode := __NEW(XOR_UINT);
Clone := pNode^;
END_METHOD

METHOD PROTECTED OnExecute
VAR
END_VAR
out.Value := in1.Value XOR in2.Value;
END_METHOD

END_FUNCTION_BLOCK

// Logic/Nodes/XOR/XOR_ULINT
{attribute 'linkalways'} 
{attribute 'no_explicit_call' := 'This FB is a CLASS and must be accessed using methods or properties'}
{attribute 'enable_dynamic_creation'}
FUNCTION_BLOCK FINAL XOR_ULINT EXTENDS Node
VAR
	in1 : _ULINT(0);
	in2 : _ULINT(0);
	out : _ULINT(0);
END_VAR

METHOD FB_init : BOOL
VAR_INPUT
	bInitRetains : BOOL; // if TRUE, the retain variables are initialized (warm start / cold start)
	bInCopyCode : BOOL;  // if TRUE, the instance afterwards gets moved into the copy code (online change)
END_VAR
AddInput('in1',THIS^.in1);
AddInput('in2',THIS^.in2);
AddOutput('out', THIS^.out);
END_METHOD

METHOD PUBLIC Clone : I_Node
VAR
	pNode : POINTER TO XOR_ULINT;
END_VAR
pNode := __NEW(XOR_ULINT);
Clone := pNode^;
END_METHOD

METHOD PROTECTED OnExecute
VAR
END_VAR
out.Value := in1.Value XOR in2.Value;
END_METHOD

END_FUNCTION_BLOCK

// Logic/Nodes/XOR/XOR_USINT
{attribute 'linkalways'} 
{attribute 'no_explicit_call' := 'This FB is a CLASS and must be accessed using methods or properties'}
{attribute 'enable_dynamic_creation'}
FUNCTION_BLOCK FINAL XOR_USINT EXTENDS Node
VAR
	in1 : _USINT(0);
	in2 : _USINT(0);
	out : _USINT(0);
END_VAR

METHOD FB_init : BOOL
VAR_INPUT
	bInitRetains : BOOL; // if TRUE, the retain variables are initialized (warm start / cold start)
	bInCopyCode : BOOL;  // if TRUE, the instance afterwards gets moved into the copy code (online change)
END_VAR
AddInput('in1',THIS^.in1);
AddInput('in2',THIS^.in2);
AddOutput('out', THIS^.out);
END_METHOD

METHOD PUBLIC Clone : I_Node
VAR
	pNode : POINTER TO XOR_USINT;
END_VAR
pNode := __NEW(XOR_USINT);
Clone := pNode^;
END_METHOD

METHOD PROTECTED OnExecute
VAR
END_VAR
out.Value := in1.Value XOR in2.Value;
END_METHOD

END_FUNCTION_BLOCK

// Logic/Nodes/XOR/XOR_WORD
{attribute 'linkalways'} 
{attribute 'no_explicit_call' := 'This FB is a CLASS and must be accessed using methods or properties'}
{attribute 'enable_dynamic_creation'}
FUNCTION_BLOCK FINAL XOR_WORD EXTENDS Node
VAR
	in1 : _WORD(0);
	in2 : _WORD(0);
	out : _WORD(0);
END_VAR

METHOD FB_init : BOOL
VAR_INPUT
	bInitRetains : BOOL; // if TRUE, the retain variables are initialized (warm start / cold start)
	bInCopyCode : BOOL;  // if TRUE, the instance afterwards gets moved into the copy code (online change)
END_VAR
AddInput('in1',THIS^.in1);
AddInput('in2',THIS^.in2);
AddOutput('out', THIS^.out);
END_METHOD

METHOD PUBLIC Clone : I_Node
VAR
	pNode : POINTER TO XOR_WORD;
END_VAR
pNode := __NEW(XOR_WORD);
Clone := pNode^;
END_METHOD

METHOD PROTECTED OnExecute
VAR
END_VAR
out.Value := in1.Value XOR in2.Value;
END_METHOD

END_FUNCTION_BLOCK

// Logic/MathLogicPack
{attribute 'linkalways'} 
{attribute 'no_explicit_call' := 'This FB is a CLASS and must be accessed using methods or properties'}
{attribute 'enable_dynamic_creation'}
FUNCTION_BLOCK MathLogicPack IMPLEMENTS I_GraphPack
VAR
	AND_BOOL : AND_BOOL;
	AND_BYTE : AND_BYTE;
	AND_DINT : AND_DINT;
	AND_DWORD : AND_DWORD;
	AND_INT : AND_INT;
	AND_LINT : AND_LINT;
	AND_LWORD : AND_LWORD;
	AND_SINT : AND_SINT;
	AND_UDINT : AND_UDINT;
	AND_UINT : AND_UINT;
	AND_ULINT : AND_ULINT;
	AND_USINT : AND_USINT;
	AND_WORD : AND_WORD;
	
	OR_BOOL : OR_BOOL;
	OR_BYTE : OR_BYTE;
	OR_DINT : OR_DINT;
	OR_DWORD : OR_DWORD;
	OR_INT : OR_INT;
	OR_LINT : OR_LINT;
	OR_LWORD : OR_LWORD;
	OR_SINT : OR_SINT;
	OR_UDINT : OR_UDINT;
	OR_UINT : OR_UINT;
	OR_ULINT : OR_ULINT;
	OR_USINT : OR_USINT;
	OR_WORD : OR_WORD;
	
	XOR_BOOL : XOR_BOOL;
	XOR_BYTE : XOR_BYTE;
	XOR_DINT : XOR_DINT;
	XOR_DWORD : XOR_DWORD;
	XOR_INT : XOR_INT;
	XOR_LINT : XOR_LINT;
	XOR_LWORD : XOR_LWORD;
	XOR_SINT : XOR_SINT;
	XOR_UDINT : XOR_UDINT;
	XOR_UINT : XOR_UINT;
	XOR_ULINT : XOR_ULINT;
	XOR_USINT : XOR_USINT;
	XOR_WORD : XOR_WORD;
	
	NOT_BOOL : NOT_BOOL;
	NOT_BYTE : NOT_BYTE;
	NOT_DINT : NOT_DINT;
	NOT_DWORD : NOT_DWORD;
	NOT_INT : NOT_INT;
	NOT_LINT : NOT_LINT;
	NOT_LWORD : NOT_LWORD;
	NOT_SINT : NOT_SINT;
	NOT_UDINT : NOT_UDINT;
	NOT_UINT : NOT_UINT;
	NOT_ULINT : NOT_ULINT;
	NOT_USINT : NOT_USINT;
	NOT_WORD : NOT_WORD;
END_VAR

METHOD Register
VAR_INPUT
	Datatypes : I_Datatypes;
	NodeFactory : I_NodeFactory;
END_VAR
NodeFactory.AddNodeAsPrototype('Math/Logic/AND/AND_BOOL',AND_BOOL);
NodeFactory.AddNodeAsPrototype('Math/Logic/AND/AND_BYTE',AND_BYTE);
NodeFactory.AddNodeAsPrototype('Math/Logic/AND/AND_DINT',AND_DINT);
NodeFactory.AddNodeAsPrototype('Math/Logic/AND/AND_DWORD',AND_DWORD);
NodeFactory.AddNodeAsPrototype('Math/Logic/AND/AND_INT',AND_INT);
NodeFactory.AddNodeAsPrototype('Math/Logic/AND/AND_LINT',AND_LINT);
NodeFactory.AddNodeAsPrototype('Math/Logic/AND/AND_LWORD',AND_LWORD);
NodeFactory.AddNodeAsPrototype('Math/Logic/AND/AND_SINT',AND_SINT);
NodeFactory.AddNodeAsPrototype('Math/Logic/AND/AND_UDINT',AND_UDINT);
NodeFactory.AddNodeAsPrototype('Math/Logic/AND/AND_UINT',AND_UINT);
NodeFactory.AddNodeAsPrototype('Math/Logic/AND/AND_ULINT',AND_ULINT);
NodeFactory.AddNodeAsPrototype('Math/Logic/AND/AND_USINT',AND_USINT);
NodeFactory.AddNodeAsPrototype('Math/Logic/AND/AND_WORD',AND_WORD);

NodeFactory.AddNodeAsPrototype('Math/Logic/OR/OR_BOOL',OR_BOOL);
NodeFactory.AddNodeAsPrototype('Math/Logic/OR/OR_BYTE',OR_BYTE);
NodeFactory.AddNodeAsPrototype('Math/Logic/OR/OR_DINT',OR_DINT);
NodeFactory.AddNodeAsPrototype('Math/Logic/OR/OR_DWORD',OR_DWORD);
NodeFactory.AddNodeAsPrototype('Math/Logic/OR/OR_INT',OR_INT);
NodeFactory.AddNodeAsPrototype('Math/Logic/OR/OR_LINT',OR_LINT);
NodeFactory.AddNodeAsPrototype('Math/Logic/OR/OR_LWORD',OR_LWORD);
NodeFactory.AddNodeAsPrototype('Math/Logic/OR/OR_SINT',OR_SINT);
NodeFactory.AddNodeAsPrototype('Math/Logic/OR/OR_UDINT',OR_UDINT);
NodeFactory.AddNodeAsPrototype('Math/Logic/OR/OR_UINT',OR_UINT);
NodeFactory.AddNodeAsPrototype('Math/Logic/OR/OR_ULINT',OR_ULINT);
NodeFactory.AddNodeAsPrototype('Math/Logic/OR/OR_USINT',OR_USINT);
NodeFactory.AddNodeAsPrototype('Math/Logic/OR/OR_WORD',OR_WORD);

NodeFactory.AddNodeAsPrototype('Math/Logic/XOR/XOR_BOOL',XOR_BOOL);
NodeFactory.AddNodeAsPrototype('Math/Logic/XOR/XOR_BYTE',XOR_BYTE);
NodeFactory.AddNodeAsPrototype('Math/Logic/XOR/XOR_DINT',XOR_DINT);
NodeFactory.AddNodeAsPrototype('Math/Logic/XOR/XOR_DWORD',XOR_DWORD);
NodeFactory.AddNodeAsPrototype('Math/Logic/XOR/XOR_INT',XOR_INT);
NodeFactory.AddNodeAsPrototype('Math/Logic/XOR/XOR_LINT',XOR_LINT);
NodeFactory.AddNodeAsPrototype('Math/Logic/XOR/XOR_LWORD',XOR_LWORD);
NodeFactory.AddNodeAsPrototype('Math/Logic/XOR/XOR_SINT',XOR_SINT);
NodeFactory.AddNodeAsPrototype('Math/Logic/XOR/XOR_UDINT',XOR_UDINT);
NodeFactory.AddNodeAsPrototype('Math/Logic/XOR/XOR_UINT',XOR_UINT);
NodeFactory.AddNodeAsPrototype('Math/Logic/XOR/XOR_ULINT',XOR_ULINT);
NodeFactory.AddNodeAsPrototype('Math/Logic/XOR/XOR_USINT',XOR_USINT);
NodeFactory.AddNodeAsPrototype('Math/Logic/XOR/XOR_WORD',XOR_WORD);

NodeFactory.AddNodeAsPrototype('Math/Logic/NOT/NOT_BOOL',NOT_BOOL);
NodeFactory.AddNodeAsPrototype('Math/Logic/NOT/NOT_BYTE',NOT_BYTE);
NodeFactory.AddNodeAsPrototype('Math/Logic/NOT/NOT_DINT',NOT_DINT);
NodeFactory.AddNodeAsPrototype('Math/Logic/NOT/NOT_DWORD',NOT_DWORD);
NodeFactory.AddNodeAsPrototype('Math/Logic/NOT/NOT_INT',NOT_INT);
NodeFactory.AddNodeAsPrototype('Math/Logic/NOT/NOT_LINT',NOT_LINT);
NodeFactory.AddNodeAsPrototype('Math/Logic/NOT/NOT_LWORD',NOT_LWORD);
NodeFactory.AddNodeAsPrototype('Math/Logic/NOT/NOT_SINT',NOT_SINT);
NodeFactory.AddNodeAsPrototype('Math/Logic/NOT/NOT_UDINT',NOT_UDINT);
NodeFactory.AddNodeAsPrototype('Math/Logic/NOT/NOT_UINT',NOT_UINT);
NodeFactory.AddNodeAsPrototype('Math/Logic/NOT/NOT_ULINT',NOT_ULINT);
NodeFactory.AddNodeAsPrototype('Math/Logic/NOT/NOT_USINT',NOT_USINT);
NodeFactory.AddNodeAsPrototype('Math/Logic/NOT/NOT_WORD',NOT_WORD);
END_METHOD

END_FUNCTION_BLOCK

// Selection/Nodes/MAX/MAX_BYTE
{attribute 'linkalways'} 
{attribute 'no_explicit_call' := 'This FB is a CLASS and must be accessed using methods or properties'}
{attribute 'enable_dynamic_creation'}
FUNCTION_BLOCK FINAL MAX_BYTE EXTENDS Node
VAR
	in1 : _BYTE(0);
	in2 : _BYTE(0);
	out : _BYTE(0);
END_VAR

METHOD FB_init : BOOL
VAR_INPUT
	bInitRetains : BOOL; // if TRUE, the retain variables are initialized (warm start / cold start)
	bInCopyCode : BOOL;  // if TRUE, the instance afterwards gets moved into the copy code (online change)
END_VAR
AddInput('in1',THIS^.in1);
AddInput('in2',THIS^.in2);
AddOutput('out', THIS^.out);
END_METHOD

METHOD PUBLIC Clone : I_Node
VAR
	pNode : POINTER TO MAX_BYTE;
END_VAR
pNode := __NEW(MAX_BYTE);
Clone := pNode^;
END_METHOD

METHOD PROTECTED OnExecute
VAR
END_VAR
out.Value := MAX(in1.Value, in2.Value);
END_METHOD

END_FUNCTION_BLOCK

// Selection/Nodes/MAX/MAX_DINT
{attribute 'linkalways'} 
{attribute 'no_explicit_call' := 'This FB is a CLASS and must be accessed using methods or properties'}
{attribute 'enable_dynamic_creation'}
FUNCTION_BLOCK FINAL MAX_DINT EXTENDS Node
VAR
	in1 : _DINT(0);
	in2 : _DINT(0);
	out : _DINT(0);
END_VAR

METHOD FB_init : BOOL
VAR_INPUT
	bInitRetains : BOOL; // if TRUE, the retain variables are initialized (warm start / cold start)
	bInCopyCode : BOOL;  // if TRUE, the instance afterwards gets moved into the copy code (online change)
END_VAR
AddInput('in1',THIS^.in1);
AddInput('in2',THIS^.in2);
AddOutput('out', THIS^.out);
END_METHOD

METHOD PUBLIC Clone : I_Node
VAR
	pNode : POINTER TO MAX_DINT;
END_VAR
pNode := __NEW(MAX_DINT);
Clone := pNode^;
END_METHOD

METHOD PROTECTED OnExecute
VAR
END_VAR
out.Value := MAX(in1.Value, in2.Value);
END_METHOD

END_FUNCTION_BLOCK

// Selection/Nodes/MAX/MAX_DWORD
{attribute 'linkalways'} 
{attribute 'no_explicit_call' := 'This FB is a CLASS and must be accessed using methods or properties'}
{attribute 'enable_dynamic_creation'}
FUNCTION_BLOCK FINAL MAX_DWORD EXTENDS Node
VAR
	in1 : _DWORD(0);
	in2 : _DWORD(0);
	out : _DWORD(0);
END_VAR

METHOD FB_init : BOOL
VAR_INPUT
	bInitRetains : BOOL; // if TRUE, the retain variables are initialized (warm start / cold start)
	bInCopyCode : BOOL;  // if TRUE, the instance afterwards gets moved into the copy code (online change)
END_VAR
AddInput('in1',THIS^.in1);
AddInput('in2',THIS^.in2);
AddOutput('out', THIS^.out);
END_METHOD

METHOD PUBLIC Clone : I_Node
VAR
	pNode : POINTER TO MAX_DWORD;
END_VAR
pNode := __NEW(MAX_DWORD);
Clone := pNode^;
END_METHOD

METHOD PROTECTED OnExecute
VAR
END_VAR
out.Value := MAX(in1.Value, in2.Value);
END_METHOD

END_FUNCTION_BLOCK

// Selection/Nodes/MAX/MAX_INT
{attribute 'linkalways'} 
{attribute 'no_explicit_call' := 'This FB is a CLASS and must be accessed using methods or properties'}
{attribute 'enable_dynamic_creation'}
FUNCTION_BLOCK FINAL MAX_INT EXTENDS Node
VAR
	in1 : _INT(0);
	in2 : _INT(0);
	out : _INT(0);
END_VAR

METHOD FB_init : BOOL
VAR_INPUT
	bInitRetains : BOOL; // if TRUE, the retain variables are initialized (warm start / cold start)
	bInCopyCode : BOOL;  // if TRUE, the instance afterwards gets moved into the copy code (online change)
END_VAR
AddInput('in1',THIS^.in1);
AddInput('in2',THIS^.in2);
AddOutput('out', THIS^.out);
END_METHOD

METHOD PUBLIC Clone : I_Node
VAR
	pNode : POINTER TO MAX_INT;
END_VAR
pNode := __NEW(MAX_INT);
Clone := pNode^;
END_METHOD

METHOD PROTECTED OnExecute
VAR
END_VAR
out.Value := MAX(in1.Value, in2.Value);
END_METHOD

END_FUNCTION_BLOCK

// Selection/Nodes/MAX/MAX_LINT
{attribute 'linkalways'} 
{attribute 'no_explicit_call' := 'This FB is a CLASS and must be accessed using methods or properties'}
{attribute 'enable_dynamic_creation'}
FUNCTION_BLOCK FINAL MAX_LINT EXTENDS Node
VAR
	in1 : _LINT(0);
	in2 : _LINT(0);
	out : _LINT(0);
END_VAR

METHOD FB_init : BOOL
VAR_INPUT
	bInitRetains : BOOL; // if TRUE, the retain variables are initialized (warm start / cold start)
	bInCopyCode : BOOL;  // if TRUE, the instance afterwards gets moved into the copy code (online change)
END_VAR
AddInput('in1',THIS^.in1);
AddInput('in2',THIS^.in2);
AddOutput('out', THIS^.out);
END_METHOD

METHOD PUBLIC Clone : I_Node
VAR
	pNode : POINTER TO MAX_LINT;
END_VAR
pNode := __NEW(MAX_LINT);
Clone := pNode^;
END_METHOD

METHOD PROTECTED OnExecute
VAR
END_VAR
out.Value := MAX(in1.Value, in2.Value);
END_METHOD

END_FUNCTION_BLOCK

// Selection/Nodes/MAX/MAX_LREAL
{attribute 'linkalways'} 
{attribute 'no_explicit_call' := 'This FB is a CLASS and must be accessed using methods or properties'}
{attribute 'enable_dynamic_creation'}
FUNCTION_BLOCK FINAL MAX_LREAL EXTENDS Node
VAR
	in1 : _LREAL(0.0);
	in2 : _LREAL(0.0);
	out : _LREAL(0.0);
END_VAR

METHOD FB_init : BOOL
VAR_INPUT
	bInitRetains : BOOL; // if TRUE, the retain variables are initialized (warm start / cold start)
	bInCopyCode : BOOL;  // if TRUE, the instance afterwards gets moved into the copy code (online change)
END_VAR
AddInput('in1',THIS^.in1);
AddInput('in2',THIS^.in2);
AddOutput('out', THIS^.out);
END_METHOD

METHOD PUBLIC Clone : I_Node
VAR
	pNode : POINTER TO MAX_LREAL;
END_VAR
pNode := __NEW(MAX_LREAL);
Clone := pNode^;
END_METHOD

METHOD PROTECTED OnExecute
VAR
END_VAR
out.Value := MAX(in1.Value, in2.Value);
END_METHOD

END_FUNCTION_BLOCK

// Selection/Nodes/MAX/MAX_LWORD
{attribute 'linkalways'} 
{attribute 'no_explicit_call' := 'This FB is a CLASS and must be accessed using methods or properties'}
{attribute 'enable_dynamic_creation'}
FUNCTION_BLOCK FINAL MAX_LWORD EXTENDS Node
VAR
	in1 : _LWORD(0);
	in2 : _LWORD(0);
	out : _LWORD(0);
END_VAR

METHOD FB_init : BOOL
VAR_INPUT
	bInitRetains : BOOL; // if TRUE, the retain variables are initialized (warm start / cold start)
	bInCopyCode : BOOL;  // if TRUE, the instance afterwards gets moved into the copy code (online change)
END_VAR
AddInput('in1',THIS^.in1);
AddInput('in2',THIS^.in2);
AddOutput('out', THIS^.out);
END_METHOD

METHOD PUBLIC Clone : I_Node
VAR
	pNode : POINTER TO MAX_LWORD;
END_VAR
pNode := __NEW(MAX_LWORD);
Clone := pNode^;
END_METHOD

METHOD PROTECTED OnExecute
VAR
END_VAR
out.Value := MAX(in1.Value, in2.Value);
END_METHOD

END_FUNCTION_BLOCK

// Selection/Nodes/MAX/MAX_REAL
{attribute 'linkalways'} 
{attribute 'no_explicit_call' := 'This FB is a CLASS and must be accessed using methods or properties'}
{attribute 'enable_dynamic_creation'}
FUNCTION_BLOCK FINAL MAX_REAL EXTENDS Node
VAR
	in1 : _REAL(0.0);
	in2 : _REAL(0.0);
	out : _REAL(0.0);
END_VAR

METHOD FB_init : BOOL
VAR_INPUT
	bInitRetains : BOOL; // if TRUE, the retain variables are initialized (warm start / cold start)
	bInCopyCode : BOOL;  // if TRUE, the instance afterwards gets moved into the copy code (online change)
END_VAR
AddInput('in1',THIS^.in1);
AddInput('in2',THIS^.in2);
AddOutput('out', THIS^.out);
END_METHOD

METHOD PUBLIC Clone : I_Node
VAR
	pNode : POINTER TO MAX_REAL;
END_VAR
pNode := __NEW(MAX_REAL);
Clone := pNode^;
END_METHOD

METHOD PROTECTED OnExecute
VAR
END_VAR
out.Value := MAX(in1.Value, in2.Value);
END_METHOD

END_FUNCTION_BLOCK

// Selection/Nodes/MAX/MAX_SINT
{attribute 'linkalways'} 
{attribute 'no_explicit_call' := 'This FB is a CLASS and must be accessed using methods or properties'}
{attribute 'enable_dynamic_creation'}
FUNCTION_BLOCK FINAL MAX_SINT EXTENDS Node
VAR
	in1 : _SINT(0);
	in2 : _SINT(0);
	out : _SINT(0);
END_VAR

METHOD FB_init : BOOL
VAR_INPUT
	bInitRetains : BOOL; // if TRUE, the retain variables are initialized (warm start / cold start)
	bInCopyCode : BOOL;  // if TRUE, the instance afterwards gets moved into the copy code (online change)
END_VAR
AddInput('in1',THIS^.in1);
AddInput('in2',THIS^.in2);
AddOutput('out', THIS^.out);
END_METHOD

METHOD PUBLIC Clone : I_Node
VAR
	pNode : POINTER TO MAX_SINT;
END_VAR
pNode := __NEW(MAX_SINT);
Clone := pNode^;
END_METHOD

METHOD PROTECTED OnExecute
VAR
END_VAR
out.Value := MAX(in1.Value, in2.Value);
END_METHOD

END_FUNCTION_BLOCK

// Selection/Nodes/MAX/MAX_UDINT
{attribute 'linkalways'} 
{attribute 'no_explicit_call' := 'This FB is a CLASS and must be accessed using methods or properties'}
{attribute 'enable_dynamic_creation'}
FUNCTION_BLOCK FINAL MAX_UDINT EXTENDS Node
VAR
	in1 : _UDINT(0);
	in2 : _UDINT(0);
	out : _UDINT(0);
END_VAR

METHOD FB_init : BOOL
VAR_INPUT
	bInitRetains : BOOL; // if TRUE, the retain variables are initialized (warm start / cold start)
	bInCopyCode : BOOL;  // if TRUE, the instance afterwards gets moved into the copy code (online change)
END_VAR
AddInput('in1',THIS^.in1);
AddInput('in2',THIS^.in2);
AddOutput('out', THIS^.out);
END_METHOD

METHOD PUBLIC Clone : I_Node
VAR
	pNode : POINTER TO MAX_UDINT;
END_VAR
pNode := __NEW(MAX_UDINT);
Clone := pNode^;
END_METHOD

METHOD PROTECTED OnExecute
VAR
END_VAR
out.Value := MAX(in1.Value, in2.Value);
END_METHOD

END_FUNCTION_BLOCK

// Selection/Nodes/MAX/MAX_UINT
{attribute 'linkalways'} 
{attribute 'no_explicit_call' := 'This FB is a CLASS and must be accessed using methods or properties'}
{attribute 'enable_dynamic_creation'}
FUNCTION_BLOCK FINAL MAX_UINT EXTENDS Node
VAR
	in1 : _UINT(0);
	in2 : _UINT(0);
	out : _UINT(0);
END_VAR

METHOD FB_init : BOOL
VAR_INPUT
	bInitRetains : BOOL; // if TRUE, the retain variables are initialized (warm start / cold start)
	bInCopyCode : BOOL;  // if TRUE, the instance afterwards gets moved into the copy code (online change)
END_VAR
AddInput('in1',THIS^.in1);
AddInput('in2',THIS^.in2);
AddOutput('out', THIS^.out);
END_METHOD

METHOD PUBLIC Clone : I_Node
VAR
	pNode : POINTER TO MAX_UINT;
END_VAR
pNode := __NEW(MAX_UINT);
Clone := pNode^;
END_METHOD

METHOD PROTECTED OnExecute
VAR
END_VAR
out.Value := MAX(in1.Value, in2.Value);
END_METHOD

END_FUNCTION_BLOCK

// Selection/Nodes/MAX/MAX_ULINT
{attribute 'linkalways'} 
{attribute 'no_explicit_call' := 'This FB is a CLASS and must be accessed using methods or properties'}
{attribute 'enable_dynamic_creation'}
FUNCTION_BLOCK FINAL MAX_ULINT EXTENDS Node
VAR
	in1 : _ULINT(0);
	in2 : _ULINT(0);
	out : _ULINT(0);
END_VAR

METHOD FB_init : BOOL
VAR_INPUT
	bInitRetains : BOOL; // if TRUE, the retain variables are initialized (warm start / cold start)
	bInCopyCode : BOOL;  // if TRUE, the instance afterwards gets moved into the copy code (online change)
END_VAR
AddInput('in1',THIS^.in1);
AddInput('in2',THIS^.in2);
AddOutput('out', THIS^.out);
END_METHOD

METHOD PUBLIC Clone : I_Node
VAR
	pNode : POINTER TO MAX_ULINT;
END_VAR
pNode := __NEW(MAX_ULINT);
Clone := pNode^;
END_METHOD

METHOD PROTECTED OnExecute
VAR
END_VAR
out.Value := MAX(in1.Value, in2.Value);
END_METHOD

END_FUNCTION_BLOCK

// Selection/Nodes/MAX/MAX_USINT
{attribute 'linkalways'} 
{attribute 'no_explicit_call' := 'This FB is a CLASS and must be accessed using methods or properties'}
{attribute 'enable_dynamic_creation'}
FUNCTION_BLOCK FINAL MAX_USINT EXTENDS Node
VAR
	in1 : _USINT(0);
	in2 : _USINT(0);
	out : _USINT(0);
END_VAR

METHOD FB_init : BOOL
VAR_INPUT
	bInitRetains : BOOL; // if TRUE, the retain variables are initialized (warm start / cold start)
	bInCopyCode : BOOL;  // if TRUE, the instance afterwards gets moved into the copy code (online change)
END_VAR
AddInput('in1',THIS^.in1);
AddInput('in2',THIS^.in2);
AddOutput('out', THIS^.out);
END_METHOD

METHOD PUBLIC Clone : I_Node
VAR
	pNode : POINTER TO MAX_USINT;
END_VAR
pNode := __NEW(MAX_USINT);
Clone := pNode^;
END_METHOD

METHOD PROTECTED OnExecute
VAR
END_VAR
out.Value := MAX(in1.Value, in2.Value);
END_METHOD

END_FUNCTION_BLOCK

// Selection/Nodes/MAX/MAX_WORD
{attribute 'linkalways'} 
{attribute 'no_explicit_call' := 'This FB is a CLASS and must be accessed using methods or properties'}
{attribute 'enable_dynamic_creation'}
FUNCTION_BLOCK FINAL MAX_WORD EXTENDS Node
VAR
	in1 : _WORD(0);
	in2 : _WORD(0);
	out : _WORD(0);
END_VAR

METHOD FB_init : BOOL
VAR_INPUT
	bInitRetains : BOOL; // if TRUE, the retain variables are initialized (warm start / cold start)
	bInCopyCode : BOOL;  // if TRUE, the instance afterwards gets moved into the copy code (online change)
END_VAR
AddInput('in1',THIS^.in1);
AddInput('in2',THIS^.in2);
AddOutput('out', THIS^.out);
END_METHOD

METHOD PUBLIC Clone : I_Node
VAR
	pNode : POINTER TO MAX_WORD;
END_VAR
pNode := __NEW(MAX_WORD);
Clone := pNode^;
END_METHOD

METHOD PROTECTED OnExecute
VAR
END_VAR
out.Value := MAX(in1.Value, in2.Value);
END_METHOD

END_FUNCTION_BLOCK

// Selection/Nodes/MIN/MIN_BYTE
{attribute 'linkalways'} 
{attribute 'no_explicit_call' := 'This FB is a CLASS and must be accessed using methods or properties'}
{attribute 'enable_dynamic_creation'}
FUNCTION_BLOCK FINAL MIN_BYTE EXTENDS Node
VAR
	in1 : _BYTE(0);
	in2 : _BYTE(0);
	out : _BYTE(0);
END_VAR

METHOD FB_init : BOOL
VAR_INPUT
	bInitRetains : BOOL; // if TRUE, the retain variables are initialized (warm start / cold start)
	bInCopyCode : BOOL;  // if TRUE, the instance afterwards gets moved into the copy code (online change)
END_VAR
AddInput('in1',THIS^.in1);
AddInput('in2',THIS^.in2);
AddOutput('out', THIS^.out);
END_METHOD

METHOD PUBLIC Clone : I_Node
VAR
	pNode : POINTER TO MIN_BYTE;
END_VAR
pNode := __NEW(MIN_BYTE);
Clone := pNode^;
END_METHOD

METHOD PROTECTED OnExecute
VAR
END_VAR
out.Value := MIN(in1.Value, in2.Value);
END_METHOD

END_FUNCTION_BLOCK

// Selection/Nodes/MIN/MIN_DINT
{attribute 'linkalways'} 
{attribute 'no_explicit_call' := 'This FB is a CLASS and must be accessed using methods or properties'}
{attribute 'enable_dynamic_creation'}
FUNCTION_BLOCK FINAL MIN_DINT EXTENDS Node
VAR
	in1 : _DINT(0);
	in2 : _DINT(0);
	out : _DINT(0);
END_VAR

METHOD FB_init : BOOL
VAR_INPUT
	bInitRetains : BOOL; // if TRUE, the retain variables are initialized (warm start / cold start)
	bInCopyCode : BOOL;  // if TRUE, the instance afterwards gets moved into the copy code (online change)
END_VAR
AddInput('in1',THIS^.in1);
AddInput('in2',THIS^.in2);
AddOutput('out', THIS^.out);
END_METHOD

METHOD PUBLIC Clone : I_Node
VAR
	pNode : POINTER TO MIN_DINT;
END_VAR
pNode := __NEW(MIN_DINT);
Clone := pNode^;
END_METHOD

METHOD PROTECTED OnExecute
VAR
END_VAR
out.Value := MIN(in1.Value, in2.Value);
END_METHOD

END_FUNCTION_BLOCK

// Selection/Nodes/MIN/MIN_DWORD
{attribute 'linkalways'} 
{attribute 'no_explicit_call' := 'This FB is a CLASS and must be accessed using methods or properties'}
{attribute 'enable_dynamic_creation'}
FUNCTION_BLOCK FINAL MIN_DWORD EXTENDS Node
VAR
	in1 : _DWORD(0);
	in2 : _DWORD(0);
	out : _DWORD(0);
END_VAR

METHOD FB_init : BOOL
VAR_INPUT
	bInitRetains : BOOL; // if TRUE, the retain variables are initialized (warm start / cold start)
	bInCopyCode : BOOL;  // if TRUE, the instance afterwards gets moved into the copy code (online change)
END_VAR
AddInput('in1',THIS^.in1);
AddInput('in2',THIS^.in2);
AddOutput('out', THIS^.out);
END_METHOD

METHOD PUBLIC Clone : I_Node
VAR
	pNode : POINTER TO MIN_DWORD;
END_VAR
pNode := __NEW(MIN_DWORD);
Clone := pNode^;
END_METHOD

METHOD PROTECTED OnExecute
VAR
END_VAR
out.Value := MIN(in1.Value, in2.Value);
END_METHOD

END_FUNCTION_BLOCK

// Selection/Nodes/MIN/MIN_INT
{attribute 'linkalways'} 
{attribute 'no_explicit_call' := 'This FB is a CLASS and must be accessed using methods or properties'}
{attribute 'enable_dynamic_creation'}
FUNCTION_BLOCK FINAL MIN_INT EXTENDS Node
VAR
	in1 : _INT(0);
	in2 : _INT(0);
	out : _INT(0);
END_VAR

METHOD FB_init : BOOL
VAR_INPUT
	bInitRetains : BOOL; // if TRUE, the retain variables are initialized (warm start / cold start)
	bInCopyCode : BOOL;  // if TRUE, the instance afterwards gets moved into the copy code (online change)
END_VAR
AddInput('in1',THIS^.in1);
AddInput('in2',THIS^.in2);
AddOutput('out', THIS^.out);
END_METHOD

METHOD PUBLIC Clone : I_Node
VAR
	pNode : POINTER TO MIN_INT;
END_VAR
pNode := __NEW(MIN_INT);
Clone := pNode^;
END_METHOD

METHOD PROTECTED OnExecute
VAR
END_VAR
out.Value := MIN(in1.Value, in2.Value);
END_METHOD

END_FUNCTION_BLOCK

// Selection/Nodes/MIN/MIN_LINT
{attribute 'linkalways'} 
{attribute 'no_explicit_call' := 'This FB is a CLASS and must be accessed using methods or properties'}
{attribute 'enable_dynamic_creation'}
FUNCTION_BLOCK FINAL MIN_LINT EXTENDS Node
VAR
	in1 : _LINT(0);
	in2 : _LINT(0);
	out : _LINT(0);
END_VAR

METHOD FB_init : BOOL
VAR_INPUT
	bInitRetains : BOOL; // if TRUE, the retain variables are initialized (warm start / cold start)
	bInCopyCode : BOOL;  // if TRUE, the instance afterwards gets moved into the copy code (online change)
END_VAR
AddInput('in1',THIS^.in1);
AddInput('in2',THIS^.in2);
AddOutput('out', THIS^.out);
END_METHOD

METHOD PUBLIC Clone : I_Node
VAR
	pNode : POINTER TO MIN_LINT;
END_VAR
pNode := __NEW(MIN_LINT);
Clone := pNode^;
END_METHOD

METHOD PROTECTED OnExecute
VAR
END_VAR
out.Value := MIN(in1.Value, in2.Value);
END_METHOD

END_FUNCTION_BLOCK

// Selection/Nodes/MIN/MIN_LREAL
{attribute 'linkalways'} 
{attribute 'no_explicit_call' := 'This FB is a CLASS and must be accessed using methods or properties'}
{attribute 'enable_dynamic_creation'}
FUNCTION_BLOCK FINAL MIN_LREAL EXTENDS Node
VAR
	in1 : _LREAL(0.0);
	in2 : _LREAL(0.0);
	out : _LREAL(0.0);
END_VAR

METHOD FB_init : BOOL
VAR_INPUT
	bInitRetains : BOOL; // if TRUE, the retain variables are initialized (warm start / cold start)
	bInCopyCode : BOOL;  // if TRUE, the instance afterwards gets moved into the copy code (online change)
END_VAR
AddInput('in1',THIS^.in1);
AddInput('in2',THIS^.in2);
AddOutput('out', THIS^.out);
END_METHOD

METHOD PUBLIC Clone : I_Node
VAR
	pNode : POINTER TO MIN_LREAL;
END_VAR
pNode := __NEW(MIN_LREAL);
Clone := pNode^;
END_METHOD

METHOD PROTECTED OnExecute
VAR
END_VAR
out.Value := MIN(in1.Value, in2.Value);
END_METHOD

END_FUNCTION_BLOCK

// Selection/Nodes/MIN/MIN_LWORD
{attribute 'linkalways'} 
{attribute 'no_explicit_call' := 'This FB is a CLASS and must be accessed using methods or properties'}
{attribute 'enable_dynamic_creation'}
FUNCTION_BLOCK FINAL MIN_LWORD EXTENDS Node
VAR
	in1 : _LWORD(0);
	in2 : _LWORD(0);
	out : _LWORD(0);
END_VAR

METHOD FB_init : BOOL
VAR_INPUT
	bInitRetains : BOOL; // if TRUE, the retain variables are initialized (warm start / cold start)
	bInCopyCode : BOOL;  // if TRUE, the instance afterwards gets moved into the copy code (online change)
END_VAR
AddInput('in1',THIS^.in1);
AddInput('in2',THIS^.in2);
AddOutput('out', THIS^.out);
END_METHOD

METHOD PUBLIC Clone : I_Node
VAR
	pNode : POINTER TO MIN_LWORD;
END_VAR
pNode := __NEW(MIN_LWORD);
Clone := pNode^;
END_METHOD

METHOD PROTECTED OnExecute
VAR
END_VAR
out.Value := MIN(in1.Value, in2.Value);
END_METHOD

END_FUNCTION_BLOCK

// Selection/Nodes/MIN/MIN_REAL
{attribute 'linkalways'} 
{attribute 'no_explicit_call' := 'This FB is a CLASS and must be accessed using methods or properties'}
{attribute 'enable_dynamic_creation'}
FUNCTION_BLOCK FINAL MIN_REAL EXTENDS Node
VAR
	in1 : _REAL(0.0);
	in2 : _REAL(0.0);
	out : _REAL(0.0);
END_VAR

METHOD FB_init : BOOL
VAR_INPUT
	bInitRetains : BOOL; // if TRUE, the retain variables are initialized (warm start / cold start)
	bInCopyCode : BOOL;  // if TRUE, the instance afterwards gets moved into the copy code (online change)
END_VAR
AddInput('in1',THIS^.in1);
AddInput('in2',THIS^.in2);
AddOutput('out', THIS^.out);
END_METHOD

METHOD PUBLIC Clone : I_Node
VAR
	pNode : POINTER TO MIN_REAL;
END_VAR
pNode := __NEW(MIN_REAL);
Clone := pNode^;
END_METHOD

METHOD PROTECTED OnExecute
VAR
END_VAR
out.Value := MIN(in1.Value, in2.Value);
END_METHOD

END_FUNCTION_BLOCK

// Selection/Nodes/MIN/MIN_SINT
{attribute 'linkalways'} 
{attribute 'no_explicit_call' := 'This FB is a CLASS and must be accessed using methods or properties'}
{attribute 'enable_dynamic_creation'}
FUNCTION_BLOCK FINAL MIN_SINT EXTENDS Node
VAR
	in1 : _SINT(0);
	in2 : _SINT(0);
	out : _SINT(0);
END_VAR

METHOD FB_init : BOOL
VAR_INPUT
	bInitRetains : BOOL; // if TRUE, the retain variables are initialized (warm start / cold start)
	bInCopyCode : BOOL;  // if TRUE, the instance afterwards gets moved into the copy code (online change)
END_VAR
AddInput('in1',THIS^.in1);
AddInput('in2',THIS^.in2);
AddOutput('out', THIS^.out);
END_METHOD

METHOD PUBLIC Clone : I_Node
VAR
	pNode : POINTER TO MIN_SINT;
END_VAR
pNode := __NEW(MIN_SINT);
Clone := pNode^;
END_METHOD

METHOD PROTECTED OnExecute
VAR
END_VAR
out.Value := MIN(in1.Value, in2.Value);
END_METHOD

END_FUNCTION_BLOCK

// Selection/Nodes/MIN/MIN_UDINT
{attribute 'linkalways'} 
{attribute 'no_explicit_call' := 'This FB is a CLASS and must be accessed using methods or properties'}
{attribute 'enable_dynamic_creation'}
FUNCTION_BLOCK FINAL MIN_UDINT EXTENDS Node
VAR
	in1 : _UDINT(0);
	in2 : _UDINT(0);
	out : _UDINT(0);
END_VAR

METHOD FB_init : BOOL
VAR_INPUT
	bInitRetains : BOOL; // if TRUE, the retain variables are initialized (warm start / cold start)
	bInCopyCode : BOOL;  // if TRUE, the instance afterwards gets moved into the copy code (online change)
END_VAR
AddInput('in1',THIS^.in1);
AddInput('in2',THIS^.in2);
AddOutput('out', THIS^.out);
END_METHOD

METHOD PUBLIC Clone : I_Node
VAR
	pNode : POINTER TO MIN_UDINT;
END_VAR
pNode := __NEW(MIN_UDINT);
Clone := pNode^;
END_METHOD

METHOD PROTECTED OnExecute
VAR
END_VAR
out.Value := MIN(in1.Value, in2.Value);
END_METHOD

END_FUNCTION_BLOCK

// Selection/Nodes/MIN/MIN_UINT
{attribute 'linkalways'} 
{attribute 'no_explicit_call' := 'This FB is a CLASS and must be accessed using methods or properties'}
{attribute 'enable_dynamic_creation'}
FUNCTION_BLOCK FINAL MIN_UINT EXTENDS Node
VAR
	in1 : _UINT(0);
	in2 : _UINT(0);
	out : _UINT(0);
END_VAR

METHOD FB_init : BOOL
VAR_INPUT
	bInitRetains : BOOL; // if TRUE, the retain variables are initialized (warm start / cold start)
	bInCopyCode : BOOL;  // if TRUE, the instance afterwards gets moved into the copy code (online change)
END_VAR
AddInput('in1',THIS^.in1);
AddInput('in2',THIS^.in2);
AddOutput('out', THIS^.out);
END_METHOD

METHOD PUBLIC Clone : I_Node
VAR
	pNode : POINTER TO MIN_UINT;
END_VAR
pNode := __NEW(MIN_UINT);
Clone := pNode^;
END_METHOD

METHOD PROTECTED OnExecute
VAR
END_VAR
out.Value := MIN(in1.Value, in2.Value);
END_METHOD

END_FUNCTION_BLOCK

// Selection/Nodes/MIN/MIN_ULINT
{attribute 'linkalways'} 
{attribute 'no_explicit_call' := 'This FB is a CLASS and must be accessed using methods or properties'}
{attribute 'enable_dynamic_creation'}
FUNCTION_BLOCK FINAL MIN_ULINT EXTENDS Node
VAR
	in1 : _ULINT(0);
	in2 : _ULINT(0);
	out : _ULINT(0);
END_VAR

METHOD FB_init : BOOL
VAR_INPUT
	bInitRetains : BOOL; // if TRUE, the retain variables are initialized (warm start / cold start)
	bInCopyCode : BOOL;  // if TRUE, the instance afterwards gets moved into the copy code (online change)
END_VAR
AddInput('in1',THIS^.in1);
AddInput('in2',THIS^.in2);
AddOutput('out', THIS^.out);
END_METHOD

METHOD PUBLIC Clone : I_Node
VAR
	pNode : POINTER TO MIN_ULINT;
END_VAR
pNode := __NEW(MIN_ULINT);
Clone := pNode^;
END_METHOD

METHOD PROTECTED OnExecute
VAR
END_VAR
out.Value := MIN(in1.Value, in2.Value);
END_METHOD

END_FUNCTION_BLOCK

// Selection/Nodes/MIN/MIN_USINT
{attribute 'linkalways'} 
{attribute 'no_explicit_call' := 'This FB is a CLASS and must be accessed using methods or properties'}
{attribute 'enable_dynamic_creation'}
FUNCTION_BLOCK FINAL MIN_USINT EXTENDS Node
VAR
	in1 : _USINT(0);
	in2 : _USINT(0);
	out : _USINT(0);
END_VAR

METHOD FB_init : BOOL
VAR_INPUT
	bInitRetains : BOOL; // if TRUE, the retain variables are initialized (warm start / cold start)
	bInCopyCode : BOOL;  // if TRUE, the instance afterwards gets moved into the copy code (online change)
END_VAR
AddInput('in1',THIS^.in1);
AddInput('in2',THIS^.in2);
AddOutput('out', THIS^.out);
END_METHOD

METHOD PUBLIC Clone : I_Node
VAR
	pNode : POINTER TO MIN_USINT;
END_VAR
pNode := __NEW(MIN_USINT);
Clone := pNode^;
END_METHOD

METHOD PROTECTED OnExecute
VAR
END_VAR
out.Value := MIN(in1.Value, in2.Value);
END_METHOD

END_FUNCTION_BLOCK

// Selection/Nodes/MIN/MIN_WORD
{attribute 'linkalways'} 
{attribute 'no_explicit_call' := 'This FB is a CLASS and must be accessed using methods or properties'}
{attribute 'enable_dynamic_creation'}
FUNCTION_BLOCK FINAL MIN_WORD EXTENDS Node
VAR
	in1 : _WORD(0);
	in2 : _WORD(0);
	out : _WORD(0);
END_VAR

METHOD FB_init : BOOL
VAR_INPUT
	bInitRetains : BOOL; // if TRUE, the retain variables are initialized (warm start / cold start)
	bInCopyCode : BOOL;  // if TRUE, the instance afterwards gets moved into the copy code (online change)
END_VAR
AddInput('in1',THIS^.in1);
AddInput('in2',THIS^.in2);
AddOutput('out', THIS^.out);
END_METHOD

METHOD PUBLIC Clone : I_Node
VAR
	pNode : POINTER TO MIN_WORD;
END_VAR
pNode := __NEW(MIN_WORD);
Clone := pNode^;
END_METHOD

METHOD PROTECTED OnExecute
VAR
END_VAR
out.Value := MIN(in1.Value, in2.Value);
END_METHOD

END_FUNCTION_BLOCK

// Selection/Nodes/SEL/SEL_BYTE
{attribute 'linkalways'} 
{attribute 'no_explicit_call' := 'This FB is a CLASS and must be accessed using methods or properties'}
{attribute 'enable_dynamic_creation'}
FUNCTION_BLOCK FINAL SEL_BYTE EXTENDS Node
VAR
	g : _BOOL(FALSE);
	in1 : _BYTE(0);
	in2 : _BYTE(0);
	out : _BYTE(0);
END_VAR

METHOD FB_init : BOOL
VAR_INPUT
	bInitRetains : BOOL; // if TRUE, the retain variables are initialized (warm start / cold start)
	bInCopyCode : BOOL;  // if TRUE, the instance afterwards gets moved into the copy code (online change)
END_VAR
AddInput('g',THIS^.g);
AddInput('in1',THIS^.in1);
AddInput('in2',THIS^.in2);
AddOutput('out', THIS^.out);
END_METHOD

METHOD PUBLIC Clone : I_Node
VAR
	pNode : POINTER TO SEL_BYTE;
END_VAR
pNode := __NEW(SEL_BYTE);
Clone := pNode^;
END_METHOD

METHOD PROTECTED OnExecute
VAR
END_VAR
IF g.value THEN
	out.value := in2.value;
ELSE
	out.value := in1.value;
END_IF
END_METHOD

END_FUNCTION_BLOCK

// Selection/Nodes/SEL/SEL_DINT
{attribute 'linkalways'} 
{attribute 'no_explicit_call' := 'This FB is a CLASS and must be accessed using methods or properties'}
{attribute 'enable_dynamic_creation'}
FUNCTION_BLOCK FINAL SEL_DINT EXTENDS Node
VAR
	g : _BOOL(FALSE);
	in1 : _DINT(0);
	in2 : _DINT(0);
	out : _DINT(0);
END_VAR

METHOD FB_init : BOOL
VAR_INPUT
	bInitRetains : BOOL; // if TRUE, the retain variables are initialized (warm start / cold start)
	bInCopyCode : BOOL;  // if TRUE, the instance afterwards gets moved into the copy code (online change)
END_VAR
AddInput('g',THIS^.g);
AddInput('in1',THIS^.in1);
AddInput('in2',THIS^.in2);
AddOutput('out', THIS^.out);
END_METHOD

METHOD PUBLIC Clone : I_Node
VAR
	pNode : POINTER TO SEL_DINT;
END_VAR
pNode := __NEW(SEL_DINT);
Clone := pNode^;
END_METHOD

METHOD PROTECTED OnExecute
VAR
END_VAR
IF g.value THEN
	out.value := in2.value;
ELSE
	out.value := in1.value;
END_IF
END_METHOD

END_FUNCTION_BLOCK

// Selection/Nodes/SEL/SEL_DWORD
{attribute 'linkalways'} 
{attribute 'no_explicit_call' := 'This FB is a CLASS and must be accessed using methods or properties'}
{attribute 'enable_dynamic_creation'}
FUNCTION_BLOCK FINAL SEL_DWORD EXTENDS Node
VAR
	g : _BOOL(FALSE);
	in1 : _DWORD(0);
	in2 : _DWORD(0);
	out : _DWORD(0);
END_VAR

METHOD FB_init : BOOL
VAR_INPUT
	bInitRetains : BOOL; // if TRUE, the retain variables are initialized (warm start / cold start)
	bInCopyCode : BOOL;  // if TRUE, the instance afterwards gets moved into the copy code (online change)
END_VAR
AddInput('g',THIS^.g);
AddInput('in1',THIS^.in1);
AddInput('in2',THIS^.in2);
AddOutput('out', THIS^.out);
END_METHOD

METHOD PUBLIC Clone : I_Node
VAR
	pNode : POINTER TO SEL_DWORD;
END_VAR
pNode := __NEW(SEL_DWORD);
Clone := pNode^;
END_METHOD

METHOD PROTECTED OnExecute
VAR
END_VAR
IF g.value THEN
	out.value := in2.value;
ELSE
	out.value := in1.value;
END_IF
END_METHOD

END_FUNCTION_BLOCK

// Selection/Nodes/SEL/SEL_INT
{attribute 'linkalways'} 
{attribute 'no_explicit_call' := 'This FB is a CLASS and must be accessed using methods or properties'}
{attribute 'enable_dynamic_creation'}
FUNCTION_BLOCK FINAL SEL_INT EXTENDS Node
VAR
	g : _BOOL(FALSE);
	in1 : _INT(0);
	in2 : _INT(0);
	out : _INT(0);
END_VAR

METHOD FB_init : BOOL
VAR_INPUT
	bInitRetains : BOOL; // if TRUE, the retain variables are initialized (warm start / cold start)
	bInCopyCode : BOOL;  // if TRUE, the instance afterwards gets moved into the copy code (online change)
END_VAR
AddInput('g',THIS^.g);
AddInput('in1',THIS^.in1);
AddInput('in2',THIS^.in2);
AddOutput('out', THIS^.out);
END_METHOD

METHOD PUBLIC Clone : I_Node
VAR
	pNode : POINTER TO SEL_INT;
END_VAR
pNode := __NEW(SEL_INT);
Clone := pNode^;
END_METHOD

METHOD PROTECTED OnExecute
VAR
END_VAR
IF g.value THEN
	out.value := in2.value;
ELSE
	out.value := in1.value;
END_IF
END_METHOD

END_FUNCTION_BLOCK

// Selection/Nodes/SEL/SEL_LINT
{attribute 'linkalways'} 
{attribute 'no_explicit_call' := 'This FB is a CLASS and must be accessed using methods or properties'}
{attribute 'enable_dynamic_creation'}
FUNCTION_BLOCK FINAL SEL_LINT EXTENDS Node
VAR
	g : _BOOL(FALSE);
	in1 : _LINT(0);
	in2 : _LINT(0);
	out : _LINT(0);
END_VAR

METHOD FB_init : BOOL
VAR_INPUT
	bInitRetains : BOOL; // if TRUE, the retain variables are initialized (warm start / cold start)
	bInCopyCode : BOOL;  // if TRUE, the instance afterwards gets moved into the copy code (online change)
END_VAR
AddInput('g',THIS^.g);
AddInput('in1',THIS^.in1);
AddInput('in2',THIS^.in2);
AddOutput('out', THIS^.out);
END_METHOD

METHOD PUBLIC Clone : I_Node
VAR
	pNode : POINTER TO SEL_LINT;
END_VAR
pNode := __NEW(SEL_LINT);
Clone := pNode^;
END_METHOD

METHOD PROTECTED OnExecute
VAR
END_VAR
IF g.value THEN
	out.value := in2.value;
ELSE
	out.value := in1.value;
END_IF
END_METHOD

END_FUNCTION_BLOCK

// Selection/Nodes/SEL/SEL_LREAL
{attribute 'linkalways'} 
{attribute 'no_explicit_call' := 'This FB is a CLASS and must be accessed using methods or properties'}
{attribute 'enable_dynamic_creation'}
FUNCTION_BLOCK FINAL SEL_LREAL EXTENDS Node
VAR
	g : _BOOL(FALSE);
	in1 : _LREAL(0.0);
	in2 : _LREAL(0.0);
	out : _LREAL(0.0);
END_VAR

METHOD FB_init : BOOL
VAR_INPUT
	bInitRetains : BOOL; // if TRUE, the retain variables are initialized (warm start / cold start)
	bInCopyCode : BOOL;  // if TRUE, the instance afterwards gets moved into the copy code (online change)
END_VAR
AddInput('g',THIS^.g);
AddInput('in1',THIS^.in1);
AddInput('in2',THIS^.in2);
AddOutput('out', THIS^.out);
END_METHOD

METHOD PUBLIC Clone : I_Node
VAR
	pNode : POINTER TO SEL_LREAL;
END_VAR
pNode := __NEW(SEL_LREAL);
Clone := pNode^;
END_METHOD

METHOD PROTECTED OnExecute
VAR
END_VAR
IF g.value THEN
	out.value := in2.value;
ELSE
	out.value := in1.value;
END_IF
END_METHOD

END_FUNCTION_BLOCK

// Selection/Nodes/SEL/SEL_LWORD
{attribute 'linkalways'} 
{attribute 'no_explicit_call' := 'This FB is a CLASS and must be accessed using methods or properties'}
{attribute 'enable_dynamic_creation'}
FUNCTION_BLOCK FINAL SEL_LWORD EXTENDS Node
VAR
	g : _BOOL(FALSE);
	in1 : _LWORD(0);
	in2 : _LWORD(0);
	out : _LWORD(0);
END_VAR

METHOD FB_init : BOOL
VAR_INPUT
	bInitRetains : BOOL; // if TRUE, the retain variables are initialized (warm start / cold start)
	bInCopyCode : BOOL;  // if TRUE, the instance afterwards gets moved into the copy code (online change)
END_VAR
AddInput('g',THIS^.g);
AddInput('in1',THIS^.in1);
AddInput('in2',THIS^.in2);
AddOutput('out', THIS^.out);
END_METHOD

METHOD PUBLIC Clone : I_Node
VAR
	pNode : POINTER TO SEL_LWORD;
END_VAR
pNode := __NEW(SEL_LWORD);
Clone := pNode^;
END_METHOD

METHOD PROTECTED OnExecute
VAR
END_VAR
IF g.value THEN
	out.value := in2.value;
ELSE
	out.value := in1.value;
END_IF
END_METHOD

END_FUNCTION_BLOCK

// Selection/Nodes/SEL/SEL_REAL
{attribute 'linkalways'} 
{attribute 'no_explicit_call' := 'This FB is a CLASS and must be accessed using methods or properties'}
{attribute 'enable_dynamic_creation'}
FUNCTION_BLOCK FINAL SEL_REAL EXTENDS Node
VAR
	g : _BOOL(FALSE);
	in1 : _REAL(0.0);
	in2 : _REAL(0.0);
	out : _REAL(0.0);
END_VAR

METHOD FB_init : BOOL
VAR_INPUT
	bInitRetains : BOOL; // if TRUE, the retain variables are initialized (warm start / cold start)
	bInCopyCode : BOOL;  // if TRUE, the instance afterwards gets moved into the copy code (online change)
END_VAR
AddInput('g',THIS^.g);
AddInput('in1',THIS^.in1);
AddInput('in2',THIS^.in2);
AddOutput('out', THIS^.out);
END_METHOD

METHOD PUBLIC Clone : I_Node
VAR
	pNode : POINTER TO SEL_REAL;
END_VAR
pNode := __NEW(SEL_REAL);
Clone := pNode^;
END_METHOD

METHOD PROTECTED OnExecute
VAR
END_VAR
IF g.value THEN
	out.value := in2.value;
ELSE
	out.value := in1.value;
END_IF
END_METHOD

END_FUNCTION_BLOCK

// Selection/Nodes/SEL/SEL_SINT
{attribute 'linkalways'} 
{attribute 'no_explicit_call' := 'This FB is a CLASS and must be accessed using methods or properties'}
{attribute 'enable_dynamic_creation'}
FUNCTION_BLOCK FINAL SEL_SINT EXTENDS Node
VAR
	g : _BOOL(FALSE);
	in1 : _SINT(0);
	in2 : _SINT(0);
	out : _SINT(0);
END_VAR

METHOD FB_init : BOOL
VAR_INPUT
	bInitRetains : BOOL; // if TRUE, the retain variables are initialized (warm start / cold start)
	bInCopyCode : BOOL;  // if TRUE, the instance afterwards gets moved into the copy code (online change)
END_VAR
AddInput('g',THIS^.g);
AddInput('in1',THIS^.in1);
AddInput('in2',THIS^.in2);
AddOutput('out', THIS^.out);
END_METHOD

METHOD PUBLIC Clone : I_Node
VAR
	pNode : POINTER TO SEL_SINT;
END_VAR
pNode := __NEW(SEL_SINT);
Clone := pNode^;
END_METHOD

METHOD PROTECTED OnExecute
VAR
END_VAR
IF g.value THEN
	out.value := in2.value;
ELSE
	out.value := in1.value;
END_IF
END_METHOD

END_FUNCTION_BLOCK

// Selection/Nodes/SEL/SEL_UDINT
{attribute 'linkalways'} 
{attribute 'no_explicit_call' := 'This FB is a CLASS and must be accessed using methods or properties'}
{attribute 'enable_dynamic_creation'}
FUNCTION_BLOCK FINAL SEL_UDINT EXTENDS Node
VAR
	g : _BOOL(FALSE);
	in1 : _UDINT(0);
	in2 : _UDINT(0);
	out : _UDINT(0);
END_VAR

METHOD FB_init : BOOL
VAR_INPUT
	bInitRetains : BOOL; // if TRUE, the retain variables are initialized (warm start / cold start)
	bInCopyCode : BOOL;  // if TRUE, the instance afterwards gets moved into the copy code (online change)
END_VAR
AddInput('g',THIS^.g);
AddInput('in1',THIS^.in1);
AddInput('in2',THIS^.in2);
AddOutput('out', THIS^.out);
END_METHOD

METHOD PUBLIC Clone : I_Node
VAR
	pNode : POINTER TO SEL_UDINT;
END_VAR
pNode := __NEW(SEL_UDINT);
Clone := pNode^;
END_METHOD

METHOD PROTECTED OnExecute
VAR
END_VAR
IF g.value THEN
	out.value := in2.value;
ELSE
	out.value := in1.value;
END_IF
END_METHOD

END_FUNCTION_BLOCK

// Selection/Nodes/SEL/SEL_UINT
{attribute 'linkalways'} 
{attribute 'no_explicit_call' := 'This FB is a CLASS and must be accessed using methods or properties'}
{attribute 'enable_dynamic_creation'}
FUNCTION_BLOCK FINAL SEL_UINT EXTENDS Node
VAR
	g : _BOOL(FALSE);
	in1 : _UINT(0);
	in2 : _UINT(0);
	out : _UINT(0);
END_VAR

METHOD FB_init : BOOL
VAR_INPUT
	bInitRetains : BOOL; // if TRUE, the retain variables are initialized (warm start / cold start)
	bInCopyCode : BOOL;  // if TRUE, the instance afterwards gets moved into the copy code (online change)
END_VAR
AddInput('g',THIS^.g);
AddInput('in1',THIS^.in1);
AddInput('in2',THIS^.in2);
AddOutput('out', THIS^.out);
END_METHOD

METHOD PUBLIC Clone : I_Node
VAR
	pNode : POINTER TO SEL_UINT;
END_VAR
pNode := __NEW(SEL_UINT);
Clone := pNode^;
END_METHOD

METHOD PROTECTED OnExecute
VAR
END_VAR
IF g.value THEN
	out.value := in2.value;
ELSE
	out.value := in1.value;
END_IF
END_METHOD

END_FUNCTION_BLOCK

// Selection/Nodes/SEL/SEL_ULINT
{attribute 'linkalways'} 
{attribute 'no_explicit_call' := 'This FB is a CLASS and must be accessed using methods or properties'}
{attribute 'enable_dynamic_creation'}
FUNCTION_BLOCK FINAL SEL_ULINT EXTENDS Node
VAR
	g : _BOOL(FALSE);
	in1 : _ULINT(0);
	in2 : _ULINT(0);
	out : _ULINT(0);
END_VAR

METHOD FB_init : BOOL
VAR_INPUT
	bInitRetains : BOOL; // if TRUE, the retain variables are initialized (warm start / cold start)
	bInCopyCode : BOOL;  // if TRUE, the instance afterwards gets moved into the copy code (online change)
END_VAR
AddInput('g',THIS^.g);
AddInput('in1',THIS^.in1);
AddInput('in2',THIS^.in2);
AddOutput('out', THIS^.out);
END_METHOD

METHOD PUBLIC Clone : I_Node
VAR
	pNode : POINTER TO SEL_ULINT;
END_VAR
pNode := __NEW(SEL_ULINT);
Clone := pNode^;
END_METHOD

METHOD PROTECTED OnExecute
VAR
END_VAR
IF g.value THEN
	out.value := in2.value;
ELSE
	out.value := in1.value;
END_IF
END_METHOD

END_FUNCTION_BLOCK

// Selection/Nodes/SEL/SEL_USINT
{attribute 'linkalways'} 
{attribute 'no_explicit_call' := 'This FB is a CLASS and must be accessed using methods or properties'}
{attribute 'enable_dynamic_creation'}
FUNCTION_BLOCK FINAL SEL_USINT EXTENDS Node
VAR
	g : _BOOL(FALSE);
	in1 : _USINT(0);
	in2 : _USINT(0);
	out : _USINT(0);
END_VAR

METHOD FB_init : BOOL
VAR_INPUT
	bInitRetains : BOOL; // if TRUE, the retain variables are initialized (warm start / cold start)
	bInCopyCode : BOOL;  // if TRUE, the instance afterwards gets moved into the copy code (online change)
END_VAR
AddInput('g',THIS^.g);
AddInput('in1',THIS^.in1);
AddInput('in2',THIS^.in2);
AddOutput('out', THIS^.out);
END_METHOD

METHOD PUBLIC Clone : I_Node
VAR
	pNode : POINTER TO SEL_USINT;
END_VAR
pNode := __NEW(SEL_USINT);
Clone := pNode^;
END_METHOD

METHOD PROTECTED OnExecute
VAR
END_VAR
IF g.value THEN
	out.value := in2.value;
ELSE
	out.value := in1.value;
END_IF
END_METHOD

END_FUNCTION_BLOCK

// Selection/Nodes/SEL/SEL_WORD
{attribute 'linkalways'} 
{attribute 'no_explicit_call' := 'This FB is a CLASS and must be accessed using methods or properties'}
{attribute 'enable_dynamic_creation'}
FUNCTION_BLOCK FINAL SEL_WORD EXTENDS Node
VAR
	g : _BOOL(FALSE);
	in1 : _WORD(0);
	in2 : _WORD(0);
	out : _WORD(0);
END_VAR

METHOD FB_init : BOOL
VAR_INPUT
	bInitRetains : BOOL; // if TRUE, the retain variables are initialized (warm start / cold start)
	bInCopyCode : BOOL;  // if TRUE, the instance afterwards gets moved into the copy code (online change)
END_VAR
AddInput('g',THIS^.g);
AddInput('in1',THIS^.in1);
AddInput('in2',THIS^.in2);
AddOutput('out', THIS^.out);
END_METHOD

METHOD PUBLIC Clone : I_Node
VAR
	pNode : POINTER TO SEL_WORD;
END_VAR
pNode := __NEW(SEL_WORD);
Clone := pNode^;
END_METHOD

METHOD PROTECTED OnExecute
VAR
END_VAR
IF g.value THEN
	out.value := in2.value;
ELSE
	out.value := in1.value;
END_IF
END_METHOD

END_FUNCTION_BLOCK

// Selection/MathSelectionPack
{attribute 'linkalways'} 
{attribute 'no_explicit_call' := 'This FB is a CLASS and must be accessed using methods or properties'}
{attribute 'enable_dynamic_creation'}
FUNCTION_BLOCK MathSelectionPack IMPLEMENTS I_GraphPack
VAR
	MAX_BYTE : MAX_BYTE;
	MAX_DINT : MAX_DINT;
	MAX_DWORD : MAX_DWORD;
	MAX_INT : MAX_INT;
	MAX_LINT : MAX_LINT;
	MAX_LREAL : MAX_LREAL;
	MAX_LWORD : MAX_LWORD;
	MAX_REAL : MAX_REAL;
	MAX_SINT : MAX_SINT;
	MAX_UDINT : MAX_UDINT;
	MAX_UINT : MAX_UINT;
	MAX_ULINT : MAX_ULINT;
	MAX_USINT : MAX_USINT;
	MAX_WORD : MAX_WORD;
	
	MIN_BYTE : MIN_BYTE;
	MIN_DINT : MIN_DINT;
	MIN_DWORD : MIN_DWORD;
	MIN_INT : MIN_INT;
	MIN_LINT : MIN_LINT;
	MIN_LREAL : MIN_LREAL;
	MIN_LWORD : MIN_LWORD;
	MIN_REAL : MIN_REAL;
	MIN_SINT : MIN_SINT;
	MIN_UDINT : MIN_UDINT;
	MIN_UINT : MIN_UINT;
	MIN_ULINT : MIN_ULINT;
	MIN_USINT : MIN_USINT;
	MIN_WORD : MIN_WORD;
	
	SEL_BYTE : SEL_BYTE;
	SEL_DINT : SEL_DINT;
	SEL_DWORD : SEL_DWORD;
	SEL_INT : SEL_INT;
	SEL_LINT : SEL_LINT;
	SEL_LREAL : SEL_LREAL;
	SEL_LWORD : SEL_LWORD;
	SEL_REAL : SEL_REAL;
	SEL_SINT : SEL_SINT;
	SEL_UDINT : SEL_UDINT;
	SEL_UINT : SEL_UINT;
	SEL_ULINT : SEL_ULINT;
	SEL_USINT : SEL_USINT;
	SEL_WORD : SEL_WORD;
END_VAR

METHOD Register
VAR_INPUT
	Datatypes : I_Datatypes;
	NodeFactory : I_NodeFactory;
END_VAR
NodeFactory.AddNodeAsPrototype('Math/Selection/MAX/MAX_BYTE',MAX_BYTE);
NodeFactory.AddNodeAsPrototype('Math/Selection/MAX/MAX_DINT',MAX_DINT);
NodeFactory.AddNodeAsPrototype('Math/Selection/MAX/MAX_DWORD',MAX_DWORD);
NodeFactory.AddNodeAsPrototype('Math/Selection/MAX/MAX_INT',MAX_INT);
NodeFactory.AddNodeAsPrototype('Math/Selection/MAX/MAX_LINT',MAX_LINT);
NodeFactory.AddNodeAsPrototype('Math/Selection/MAX/MAX_LREAL',MAX_LREAL);
NodeFactory.AddNodeAsPrototype('Math/Selection/MAX/MAX_LWORD',MAX_LWORD);
NodeFactory.AddNodeAsPrototype('Math/Selection/MAX/MAX_REAL',MAX_REAL);
NodeFactory.AddNodeAsPrototype('Math/Selection/MAX/MAX_SINT',MAX_SINT);
NodeFactory.AddNodeAsPrototype('Math/Selection/MAX/MAX_UDINT',MAX_UDINT);
NodeFactory.AddNodeAsPrototype('Math/Selection/MAX/MAX_UINT',MAX_UINT);
NodeFactory.AddNodeAsPrototype('Math/Selection/MAX/MAX_ULINT',MAX_ULINT);
NodeFactory.AddNodeAsPrototype('Math/Selection/MAX/MAX_USINT',MAX_USINT);
NodeFactory.AddNodeAsPrototype('Math/Selection/MAX/MAX_WORD',MAX_WORD);

NodeFactory.AddNodeAsPrototype('Math/Selection/MIN/MIN_BYTE',MIN_BYTE);
NodeFactory.AddNodeAsPrototype('Math/Selection/MIN/MIN_DINT',MIN_DINT);
NodeFactory.AddNodeAsPrototype('Math/Selection/MIN/MIN_DWORD',MIN_DWORD);
NodeFactory.AddNodeAsPrototype('Math/Selection/MIN/MIN_INT',MIN_INT);
NodeFactory.AddNodeAsPrototype('Math/Selection/MIN/MIN_LINT',MIN_LINT);
NodeFactory.AddNodeAsPrototype('Math/Selection/MIN/MIN_LREAL',MIN_LREAL);
NodeFactory.AddNodeAsPrototype('Math/Selection/MIN/MIN_LWORD',MIN_LWORD);
NodeFactory.AddNodeAsPrototype('Math/Selection/MIN/MIN_REAL',MIN_REAL);
NodeFactory.AddNodeAsPrototype('Math/Selection/MIN/MIN_SINT',MIN_SINT);
NodeFactory.AddNodeAsPrototype('Math/Selection/MIN/MIN_UDINT',MIN_UDINT);
NodeFactory.AddNodeAsPrototype('Math/Selection/MIN/MIN_UINT',MIN_UINT);
NodeFactory.AddNodeAsPrototype('Math/Selection/MIN/MIN_ULINT',MIN_ULINT);
NodeFactory.AddNodeAsPrototype('Math/Selection/MIN/MIN_USINT',MIN_USINT);
NodeFactory.AddNodeAsPrototype('Math/Selection/MIN/MIN_WORD',MIN_WORD);

NodeFactory.AddNodeAsPrototype('Math/Selection/SEL/SEL_BYTE',SEL_BYTE);
NodeFactory.AddNodeAsPrototype('Math/Selection/SEL/SEL_DINT',SEL_DINT);
NodeFactory.AddNodeAsPrototype('Math/Selection/SEL/SEL_DWORD',SEL_DWORD);
NodeFactory.AddNodeAsPrototype('Math/Selection/SEL/SEL_INT',SEL_INT);
NodeFactory.AddNodeAsPrototype('Math/Selection/SEL/SEL_LINT',SEL_LINT);
NodeFactory.AddNodeAsPrototype('Math/Selection/SEL/SEL_LREAL',SEL_LREAL);
NodeFactory.AddNodeAsPrototype('Math/Selection/SEL/SEL_LWORD',SEL_LWORD);
NodeFactory.AddNodeAsPrototype('Math/Selection/SEL/SEL_REAL',SEL_REAL);
NodeFactory.AddNodeAsPrototype('Math/Selection/SEL/SEL_SINT',SEL_SINT);
NodeFactory.AddNodeAsPrototype('Math/Selection/SEL/SEL_UDINT',SEL_UDINT);
NodeFactory.AddNodeAsPrototype('Math/Selection/SEL/SEL_UINT',SEL_UINT);
NodeFactory.AddNodeAsPrototype('Math/Selection/SEL/SEL_ULINT',SEL_ULINT);
NodeFactory.AddNodeAsPrototype('Math/Selection/SEL/SEL_USINT',SEL_USINT);
NodeFactory.AddNodeAsPrototype('Math/Selection/SEL/SEL_WORD',SEL_WORD);
END_METHOD

END_FUNCTION_BLOCK

// MathPack
{attribute 'linkalways'} 
{attribute 'no_explicit_call' := 'This FB is a CLASS and must be accessed using methods or properties'}
{attribute 'enable_dynamic_creation'}
FUNCTION_BLOCK MathPack IMPLEMENTS I_GraphPack
VAR
	mathCorePack : MathCorePack;
	mathLogicPack : MathLogicPack;
	mathAdvancedPack : MathAdvancedPack;
	mathComparisonPack : MathComparisonPack;
	mathSelectionPack : MathSelectionPack;
END_VAR

METHOD Register
VAR_INPUT
	Datatypes : I_Datatypes;
	NodeFactory : I_NodeFactory;
END_VAR
mathCorePack.Register(Datatypes, NodeFactory);
mathLogicPack.Register(Datatypes, NodeFactory);
mathAdvancedPack.Register(Datatypes, NodeFactory);
mathComparisonPack.Register(Datatypes, NodeFactory);
mathSelectionPack.Register(Datatypes, NodeFactory);
END_METHOD

END_FUNCTION_BLOCK
